    IF (_eMessageLevel = E_MessageType.eMessageVerbose)
    THEN
      _stMsg.eType            := E_MessageType.eMessageVerbose;
      _stMsg.eSubdevice       := e_Subdevice.fbHalt;
      _stMsg.iErrorNumber     := _nErrorId;
      _stMsg.sText            := TO_STRING(_eState);
      f_MessageSet(_stMsg, _nXpu);
    END_IF
END_CASE
//-----------------------------------------------------------------------------
//-----------------------------------------------------------------------------
CASE _eState
OF
  E_PROGRESS.PROGRESS_PREPARE:
    _fbHalt(Axis              := _Mover, 
            Execute           := TRUE, 
            Deceleration      := stMoveData.rAcc, 
            Jerk              := stMoveData.rJerk, 
            BufferMode        := Tc2_MC2.MC_BufferMode.MC_Aborting);

    IF _fbHalt.Error
    THEN
      _bError                 := TRUE;
      _nErrorId               := _fbHalt.ErrorID;
      _eState                 := E_PROGRESS.PROGRESS_ERROR;

      _stMsg.eType            := E_MessageType.eMessageError;
      _stMsg.eSubdevice       := e_Subdevice.fbHalt;
      _stMsg.iErrorNumber     := _nErrorId;
      _stMsg.sText            := TO_STRING(_eState);
      f_MessageSet(_stMsg, _nXpu);

    ELSIF NOT _Mover.Status.Moving
    THEN
      _eState                 := E_PROGRESS.PROGRESS_DONE;

      IF (_eMessageLevel > E_MessageType.eMessageError)
      THEN
        _stMsg.eType          := E_MessageType.eMessageInfo;
        _stMsg.eSubdevice     := e_Subdevice.fbHalt;
        _stMsg.iErrorNumber   := _nErrorId;
        _stMsg.sText          := TO_STRING(_eState);
        f_MessageSet(_stMsg, _nXpu);
      END_IF
    END_IF
END_CASE
//-----------------------------------------------------------------------------
//-----------------------------------------------------------------------------
CASE _eState
OF
  E_PROGRESS.PROGRESS_ERROR,
  E_PROGRESS.PROGRESS_DONE:
    _stInfo.nErrorId          := _nErrorId;
    _fbHalt(
            Axis              := _Mover, 
            Execute           := FALSE);
END_CASE
//-----------------------------------------------------------------------------
//-----------------------------------------------------------------------------

Halt                          := _eState;
END_METHOD

METHOD HaltCa : E_PROGRESS
VAR_INPUT
  Execute             : BOOL;
  stMoveData          : ST_MOVE_DATA;
END_VAR
VAR_INST
  _nErrorId           : UDINT;
  _eState             : E_PROGRESS;
END_VAR
IF NOT Execute 
THEN 
	_eState := E_PROGRESS.PROGRESS_INIT; 
END_IF 
IF NOT Check() 
THEN 
	HaltCa := E_PROGRESS.PROGRESS_ERROR; 
	RETURN; 
END_IF


CASE _eState
OF
  E_PROGRESS.PROGRESS_INIT:
    IF Execute
    THEN
      _nErrorId               := 0;
      _eState                 := E_PROGRESS.PROGRESS_BUSY;
    END_IF
END_CASE
//-----------------------------------------------------------------------------
//-----------------------------------------------------------------------------
CASE _eState
OF
  E_PROGRESS.PROGRESS_BUSY:
    _eState                   := E_PROGRESS.PROGRESS_PREPARE;
    _fbHaltCa(
            Axis              := _Mover, 
            Execute           := FALSE, 
            Deceleration      := stMoveData.rAcc, 
            Jerk              := stMoveData.rJerk, 
            Gap               := stMoveData.rGap);

    IF (_eMessageLevel = E_MessageType.eMessageVerbose)
    THEN
      _stMsg.eType            := E_MessageType.eMessageVerbose;
      _stMsg.eSubdevice       := e_Subdevice.fbHaltCa;
      _stMsg.iErrorNumber     := _nErrorId;
      _stMsg.sText            := TO_STRING(_eState);
      f_MessageSet(_stMsg, _nXpu);
    END_IF
END_CASE
//-----------------------------------------------------------------------------
//-----------------------------------------------------------------------------
CASE _eState
OF
  E_PROGRESS.PROGRESS_PREPARE:
    _fbHaltCa(
            Axis              := _Mover, 
            Execute           := TRUE, 
            Deceleration      := stMoveData.rAcc, 
            Jerk              := stMoveData.rJerk, 
            Gap               := stMoveData.rGap);

    IF _fbHaltCa.Error
    THEN
      _bError                 := TRUE;
      _nErrorId               := _fbHalt.ErrorID;
      _eState                 := E_PROGRESS.PROGRESS_ERROR;

      _stMsg.eType            := E_MessageType.eMessageError;
      _stMsg.eSubdevice       := e_Subdevice.fbHaltCa;
      _stMsg.iErrorNumber     := _nErrorId;
      _stMsg.sText            := TO_STRING(_eState);
      f_MessageSet(_stMsg, _nXpu);

    ELSIF NOT _Mover.Status.Moving
    THEN
      _eState                 := E_PROGRESS.PROGRESS_DONE;

      IF (_eMessageLevel > E_MessageType.eMessageError)
      THEN
        _stMsg.eType          := E_MessageType.eMessageInfo;
        _stMsg.eSubdevice     := e_Subdevice.fbHaltCa;
        _stMsg.iErrorNumber   := _nErrorId;
        _stMsg.sText          := TO_STRING(_eState);
        f_MessageSet(_stMsg, _nXpu);
      END_IF
    END_IF
END_CASE
//-----------------------------------------------------------------------------
//-----------------------------------------------------------------------------
CASE _eState
OF
  E_PROGRESS.PROGRESS_ERROR,
  E_PROGRESS.PROGRESS_DONE:
    _stInfo.nErrorId          := _nErrorId;
    _fbHaltCa(
            Axis              := _Mover, 
            Execute           := FALSE);
END_CASE
//-----------------------------------------------------------------------------
//-----------------------------------------------------------------------------

HaltCa                          := _eState;
END_METHOD

PROPERTY LastGap : REFERENCE to lreal
SET
_rLastGap REF= LastGap;
END_SET
END_PROPERTY

PROPERTY LastPosition : REFERENCE to LREAL
SET
_rLastPosition REF= LastPosition;
END_SET
END_PROPERTY

PROPERTY Master : REFERENCE to AXIS_REF
SET
_Master REF= Master;
END_SET
END_PROPERTY

PROPERTY MessageLevel : e_messagetype
SET
_eMessageLevel := MessageLevel;
END_SET
END_PROPERTY

PROPERTY ModuloTurn : dint
GET
ModuloTurn := _Mover.NcToPlc.ModuloSetTurns;
END_GET
END_PROPERTY

PROPERTY Mover : REFERENCE to AXIS_REF
SET
_Mover REF= Mover;
END_SET
END_PROPERTY

PROPERTY MoverId : uint
SET
_nMoverId := MoverId;
END_SET
END_PROPERTY

PROPERTY MoverInfo : REFERENCE to ST_MOVER_INFO
SET


	_stInfo ref= MoverInfo;
END_SET
END_PROPERTY

METHOD MoveToPos : E_PROGRESS
VAR_INPUT
  Execute             : BOOL;
  stMoveData          : ST_MOVE_DATA;
END_VAR
VAR_INST
  _nErrorId           : UDINT;
  _rDelta,
  _rPos               : LREAL;
  _eState             : E_PROGRESS;
END_VAR
IF NOT Execute THEN _eState  := E_PROGRESS.PROGRESS_INIT; END_IF 
IF NOT Check() THEN MoveToPos   := E_PROGRESS.PROGRESS_ERROR; RETURN; END_IF


CASE _eState
OF
  E_PROGRESS.PROGRESS_INIT:
    IF Execute
    THEN
      _nErrorId               := 0;
      _rDelta                 := SEL((stMoveData.rDelta < 0.01), stMoveData.rDelta, 0.05);
      _eState                 := E_PROGRESS.PROGRESS_BUSY;
    END_IF
END_CASE
//-----------------------------------------------------------------------------
//-----------------------------------------------------------------------------
CASE _eState
OF
  E_PROGRESS.PROGRESS_BUSY:
    _eState                   := E_PROGRESS.PROGRESS_PREPARE;
    _fbPower.Override         := stMoveData.rOverride;

    _rPos                     := ABS(_Mover.NcToPlc.ModuloActTurns)* _RailLength + stMoveData.rPos;


    _rLastPosition            := _rPos;
    //_rLastGap                 := stMoveData.rGap;

    _fbMoveAbs(
            Axis              := _Mover, 
            Execute           := FALSE, 
            Position          := _rPos, 
            Velocity          := stMoveData.rVelo, 
            Acceleration      := stMoveData.rAcc, 
            Deceleration      := stMoveData.rAcc, 
            Jerk              := stMoveData.rJerk, 
            BufferMode        := Tc2_MC2.MC_BufferMode.MC_Aborting);

      IF (_eMessageLevel = E_MessageType.eMessageVerbose)
      THEN
        _stMsg.eType          := E_MessageType.eMessageVerbose;
        _stMsg.eSubdevice     := e_Subdevice.fbMovePtP;
        _stMsg.iErrorNumber   := _nErrorId;
        _stMsg.sText          := concat(TO_STRING(_eState), ': ');
        _stMsg.sText          := concat(_stMsg.sText, concat('stMoveData.rPos: ', TO_STRING(stMoveData.rPos)));
        f_MessageSet(_stMsg, _nXpu);
      END_IF
END_CASE
//-----------------------------------------------------------------------------
//-----------------------------------------------------------------------------
CASE _eState
OF
  E_PROGRESS.PROGRESS_PREPARE:
    _fbMoveAbs(
            Axis              := _Mover, 
            Execute           := TRUE, 
            Position          := _rPos, 
            Velocity          := stMoveData.rVelo, 
            Acceleration      := stMoveData.rAcc, 
            Deceleration      := stMoveData.rAcc, 
            Jerk              := stMoveData.rJerk, 
            BufferMode        := Tc2_MC2.MC_BufferMode.MC_Aborting);

    IF _fbMoveAbs.Error
    THEN
      _bError                 := TRUE;
      _nErrorId               := _fbMoveAbs.ErrorId;
      _eState                 := E_PROGRESS.PROGRESS_ERROR;

      _stMsg.eType            := E_MessageType.eMessageError;
      _stMsg.eSubdevice       := e_Subdevice.fbMovePtP;
      _stMsg.iErrorNumber     := _nErrorId;
      _stMsg.sText            := TO_STRING(_eState);
      f_MessageSet(_stMsg, _nXpu);

    ELSIF _fbMoveAbs.Active OR 
          _fbMoveAbs.Done
		THEN
      _eState                 := E_PROGRESS.PROGRESS_WORKING;

      IF (_eMessageLevel = E_MessageType.eMessageVerbose)
      THEN
        _stMsg.eType          := E_MessageType.eMessageVerbose;
        _stMsg.eSubdevice     := e_Subdevice.fbMovePtP;
        _stMsg.iErrorNumber   := _nErrorId;
        _stMsg.sText          := concat(TO_STRING(_eState), ': ');
        _stMsg.sText          := concat(_stMsg.sText, '.ModuloActPos: ');
        _stMsg.sText          := concat(_stMsg.sText, TO_STRING(_Mover.NcToPlc.ModuloActPos));
        f_MessageSet(_stMsg, _nXpu);
      END_IF
    END_IF
END_CASE
//-----------------------------------------------------------------------------
//-----------------------------------------------------------------------------
CASE _eState
OF
  E_PROGRESS.PROGRESS_WORKING:
    _fbMoveAbs(
          Axis                := _Mover);

    IF _fbMoveAbs.Error
    THEN
      _bError                 := TRUE;
      _nErrorId               := _fbMoveAbs.ErrorId;
      _stInfo.nErrorId        := _nErrorId;
      _eState                 := E_PROGRESS.PROGRESS_ERROR;

      _stMsg.eType            := E_MessageType.eMessageError;
      _stMsg.eSubdevice       := e_Subdevice.fbMovePtP;
      _stMsg.iErrorNumber     := _nErrorId;
      _stMsg.sText            := TO_STRING(_eState);
      f_MessageSet(_stMsg, _nXpu);

      _fbMoveAbs( 
            Axis              := _Mover, 
            Execute           := FALSE);


    ELSIF (_Mover.NcToPlc.ActPos > _fbMoveAbs.Position - _rDelta) AND
          (_Mover.NcToPlc.ActPos < _fbMoveAbs.Position + _rDelta)
    THEN
      IF NOT _Mover.Status.Moving
      THEN
        _eState               := E_PROGRESS.PROGRESS_DONE;

        IF (_eMessageLevel > E_MessageType.eMessageError)
        THEN
          _stMsg.eType        := E_MessageType.eMessageInfo;
          _stMsg.eSubdevice   := e_Subdevice.fbMovePtP;
          _stMsg.iErrorNumber := _nErrorId;
          _stMsg.sText        := concat(TO_STRING(_eState), ': ');
          _stMsg.sText        := concat(_stMsg.sText, concat('ModActPos: ', TO_STRING(_Mover.NcToPlc.ModuloActPos)));
          f_MessageSet(_stMsg, _nXpu);
        END_IF
      _fbMoveAbs( 
            Axis              := _Mover, 
            Execute           := FALSE);
      END_IF
    END_IF
END_CASE
//-----------------------------------------------------------------------------
//-----------------------------------------------------------------------------

MoveToPos                   := _eState;
END_METHOD

METHOD MoveToPosCa : E_PROGRESS
VAR_INPUT
  Execute             : BOOL;
  stMoveData          : ST_MOVE_DATA;
END_VAR
VAR_INST
  _nErrorId           : UDINT;
  _rDelta,
  _rPos               : LREAL;
  _eState             : E_PROGRESS;
END_VAR
IF NOT Execute THEN _eState  := E_PROGRESS.PROGRESS_INIT; END_IF 
IF NOT Check() THEN MoveToPosCa   := E_PROGRESS.PROGRESS_ERROR; RETURN; END_IF


CASE _eState
OF
  E_PROGRESS.PROGRESS_INIT:
    IF Execute
    THEN
      _nErrorId               := 0;
      _rDelta                 := SEL((stMoveData.rDelta < 0.01), stMoveData.rDelta, 0.05);
      _eState                 := E_PROGRESS.PROGRESS_BUSY;
    END_IF
END_CASE
//-----------------------------------------------------------------------------
//-----------------------------------------------------------------------------
CASE _eState
OF
  E_PROGRESS.PROGRESS_BUSY:
    _eState                   := E_PROGRESS.PROGRESS_PREPARE;
    _fbPower.Override         := stMoveData.rOverride;

    _rPos                     := ABS(_Mover.NcToPlc.ModuloActTurns)* _RailLength + stMoveData.rPos;


    _rLastPosition            := _rPos;
    _rLastGap                 := stMoveData.rGap;

    _fbMoveAbsCa( 
            Axis              := _Mover, 
            Execute           := FALSE, 
            ContinuousUpdate  := TRUE, 
            Position          := _rPos,
            Velocity          := stMoveData.rVelo, 
            Acceleration      := stMoveData.rAcc, 
            Deceleration      := stMoveData.rAcc, 
            Jerk              := stMoveData.rJerk, 
            Gap               := stMoveData.rGap, 
            BufferMode        := Tc3_Mc3Definitions.MC_BUFFER_MODE.mcAborting);

    IF (_eMessageLevel = E_MessageType.eMessageVerbose)
    THEN
      _stMsg.eType            := E_MessageType.eMessageVerbose;
      _stMsg.eSubdevice       := e_Subdevice.fbMoveToPosCa;
      _stMsg.iErrorNumber     := _nErrorId;
      _stMsg.sText            := concat(TO_STRING(_eState), ': ');
      _stMsg.sText            := concat(_stMsg.sText, concat('stMoveData.rPos: ', TO_STRING(stMoveData.rPos)));
      f_MessageSet(_stMsg, _nXpu);
    END_IF
END_CASE
//-----------------------------------------------------------------------------
//-----------------------------------------------------------------------------
CASE _eState
OF
  E_PROGRESS.PROGRESS_PREPARE:
    _fbMoveAbsCa( 
            Axis              := _Mover, 
            Execute           := TRUE, 
            ContinuousUpdate  := TRUE, 
            Position          := _rPos,
            Velocity          := stMoveData.rVelo, 
            Acceleration      := stMoveData.rAcc, 
            Deceleration      := stMoveData.rAcc, 
            Jerk              := stMoveData.rJerk, 
            Gap               := stMoveData.rGap, 
            BufferMode        := Tc3_Mc3Definitions.MC_BUFFER_MODE.mcAborting);

    IF _fbMoveAbsCa.Error
    THEN
      _bError                 := TRUE;
      _nErrorId               := _fbMoveAbsCa.ErrorId;
      _stInfo.nErrorId        := _nErrorId;
      _eState                 := E_PROGRESS.PROGRESS_ERROR;

      _stMsg.eType            := E_MessageType.eMessageError;
      _stMsg.eSubdevice       := e_Subdevice.fbMoveToPosCa;
      _stMsg.iErrorNumber     := _nErrorId;
      _stMsg.sText            := TO_STRING(_eState);
      f_MessageSet(_stMsg, _nXpu);

    ELSIF _fbMoveAbsCa.Active OR 
          _fbMoveAbsCa.Done
		THEN
      _eState                 := E_PROGRESS.PROGRESS_WORKING;

      IF (_eMessageLevel = E_MessageType.eMessageVerbose)
      THEN
        _stMsg.eType          := E_MessageType.eMessageVerbose;
        _stMsg.eSubdevice     := e_Subdevice.fbMoveToPosCa;
        _stMsg.iErrorNumber   := _nErrorId;
        _stMsg.sText          := concat(TO_STRING(_eState), ': ');
        _stMsg.sText          := concat(_stMsg.sText, '.ModuloActPos: ');
        _stMsg.sText          := concat(_stMsg.sText, TO_STRING(_Mover.NcToPlc.ModuloActPos));
        f_MessageSet(_stMsg, _nXpu);
      END_IF
    END_IF
END_CASE
//-----------------------------------------------------------------------------
//-----------------------------------------------------------------------------
CASE _eState
OF
  E_PROGRESS.PROGRESS_WORKING:
    _fbMoveAbsCa(
          Axis                := _Mover);

    IF _fbMoveAbsCa.Error
    THEN
      _bError                 := TRUE;
      _nErrorId               := _fbMoveAbsCa.ErrorId;
      _stInfo.nErrorId        := _nErrorId;
      _fbMoveAbsCa( 
            Axis              := _Mover, 
            Execute           := FALSE);

      _eState                 := E_PROGRESS.PROGRESS_ERROR;

      _stMsg.eType            := E_MessageType.eMessageError;
      _stMsg.eSubdevice       := e_Subdevice.fbMoveToPosCa;
      _stMsg.iErrorNumber     := _nErrorId;
      _stMsg.sText            := concat(TO_STRING(_eState), ': ');
      _stMsg.sText            := concat(_stMsg.sText, concat('ModActPos: ', TO_STRING(_Mover.NcToPlc.ModuloActPos)));

      f_MessageSet(_stMsg, _nXpu);

    ELSIF (_Mover.NcToPlc.ActPos > _fbMoveAbsCa.Position - _rDelta) AND
          (_Mover.NcToPlc.ActPos < _fbMoveAbsCa.Position + _rDelta)
    THEN
      IF NOT _Mover.Status.Moving
      THEN
        _eState               := E_PROGRESS.PROGRESS_DONE;

        IF (_eMessageLevel > E_MessageType.eMessageError)
        THEN
          _stMsg.eType        := E_MessageType.eMessageInfo;
          _stMsg.eSubdevice   := e_Subdevice.fbMoveToPosCa;
          _stMsg.iErrorNumber := _nErrorId;
          _stMsg.sText        := concat(TO_STRING(_eState), ': ');
          _stMsg.sText        := concat(_stMsg.sText, concat('ModActPos: ', TO_STRING(_Mover.NcToPlc.ModuloActPos)));
          f_MessageSet(_stMsg, _nXpu);
        END_IF
      _fbMoveAbsCa( 
            Axis              := _Mover, 
            Execute           := FALSE);
      END_IF
    END_IF
END_CASE
//-----------------------------------------------------------------------------
//-----------------------------------------------------------------------------

MoveToPosCa                   := _eState;
END_METHOD

PROPERTY RailLength : LREAL
GET
RailLength := _RailLength;
END_GET
SET
_RailLength := RailLength;
END_SET
END_PROPERTY

METHOD Reset : E_PROGRESS
VAR_INPUT
  Execute             : BOOL;
END_VAR
VAR_INST
  _nErrorId           : UDINT;
  _eState             : E_PROGRESS;
END_VAR
IF NOT Execute THEN _eState  := E_PROGRESS.PROGRESS_INIT; END_IF 
IF NOT Check() THEN Reset    := E_PROGRESS.PROGRESS_ERROR; RETURN; END_IF


CASE _eState
OF
  E_PROGRESS.PROGRESS_INIT:
    IF Execute
    THEN
      _stInfo.nErrorId        :=
      _nErrorId               := 0;
      _eState                 := E_PROGRESS.PROGRESS_BUSY;
    END_IF
END_CASE
//-----------------------------------------------------------------------------
//-----------------------------------------------------------------------------
CASE _eState
OF
  E_PROGRESS.PROGRESS_BUSY:
    _eState                   := E_PROGRESS.PROGRESS_PREPARE;
    _fbReset(
            Axis              := _Mover, 
            Execute           := FALSE);

    IF (_eMessageLevel = E_MessageType.eMessageVerbose)
    THEN
      _stMsg.eType            := E_MessageType.eMessageVerbose;
      _stMsg.eSubdevice       := e_Subdevice.fbReset;
      _stMsg.iErrorNumber     := _nErrorId;
      _stMsg.sText            := TO_STRING(_eState);
      f_MessageSet(_stMsg, _nXpu);
    END_IF
END_CASE
//-----------------------------------------------------------------------------
//-----------------------------------------------------------------------------
CASE _eState
OF
  E_PROGRESS.PROGRESS_PREPARE:
    _fbReset(
            Axis              := _Mover, 
            Execute           := TRUE);

    IF _fbReset.Error
    THEN
      _nErrorId               := _fbReset.ErrorID;
      _eState                 := E_PROGRESS.PROGRESS_ERROR;

      _stMsg.eType            := E_MessageType.eMessageError;
      _stMsg.eSubdevice       := e_Subdevice.fbReset;
      _stMsg.iErrorNumber     := _nErrorId;
      _stMsg.sText            := TO_STRING(_eState);
      f_MessageSet(_stMsg, _nXpu);

    ELSIF NOT _Mover.Status.Moving
    THEN
      _eState                 := E_PROGRESS.PROGRESS_DONE;

      IF (_eMessageLevel > E_MessageType.eMessageError)
      THEN
        _stMsg.eType          := E_MessageType.eMessageInfo;
        _stMsg.eSubdevice     := e_Subdevice.fbReset;
        _stMsg.iErrorNumber   := _nErrorId;
        _stMsg.sText          := TO_STRING(_eState);
        f_MessageSet(_stMsg, _nXpu);
      END_IF
    END_IF
END_CASE
//-----------------------------------------------------------------------------
//-----------------------------------------------------------------------------
CASE _eState
OF
  E_PROGRESS.PROGRESS_ERROR,
  E_PROGRESS.PROGRESS_DONE:
    _stInfo.nErrorId          := _nErrorId;
    _fbReset(
            Axis              := _Mover, 
            Execute           := FALSE);
			
	_bError := FALSE;		
END_CASE
//-----------------------------------------------------------------------------
//-----------------------------------------------------------------------------

Reset                         := _eState;
END_METHOD

METHOD SendToAbsPosCa : E_PROGRESS
VAR_INPUT
  Execute             : BOOL;
  stMoveData          : ST_MOVE_DATA;
END_VAR
VAR_INST
  _nErrorId           : UDINT;
  _rPos               : LREAL;
  _rStart             : LREAL;
  _eState             : E_PROGRESS;
END_VAR
IF NOT Execute THEN _eState  := E_PROGRESS.PROGRESS_INIT; END_IF 
IF NOT Check() THEN SendToAbsPosCa   := E_PROGRESS.PROGRESS_ERROR; RETURN; END_IF


CASE _eState
OF
  E_PROGRESS.PROGRESS_INIT:
    IF Execute
    THEN
      _nErrorId               := 0;
      _rStart                 := _Mover.NcToPlc.ActPos;

      _eState                 := E_PROGRESS.PROGRESS_BUSY;
    END_IF
END_CASE
//-----------------------------------------------------------------------------
//-----------------------------------------------------------------------------
CASE _eState
OF
  E_PROGRESS.PROGRESS_BUSY:
    _eState                   := E_PROGRESS.PROGRESS_PREPARE;
    _fbPower.Override         := stMoveData.rOverride;

    _rPos                     := stMoveData.rPos;
	
    _rLastPosition            := _rPos;
    _rLastGap                 := stMoveData.rGap;

    _fbMoveAbsCa( 
            Axis              := _Mover, 
            Execute           := FALSE, 
            ContinuousUpdate  := TRUE, 
            Position          := _rPos,
            Velocity          := stMoveData.rVelo, 
            Acceleration      := stMoveData.rAcc, 
            Deceleration      := stMoveData.rAcc, 
            Jerk              := stMoveData.rJerk, 
            Gap               := stMoveData.rGap, 
            BufferMode        := Tc3_Mc3Definitions.MC_BUFFER_MODE.mcAborting);

    IF (_eMessageLevel = E_MessageType.eMessageVerbose)
    THEN
      _stMsg.eType            := E_MessageType.eMessageVerbose;
      _stMsg.eSubdevice       := e_Subdevice.fbSendToAbsPosCa;
      _stMsg.iErrorNumber     := _nErrorId;
      _stMsg.sText            := concat(TO_STRING(_eState), ': ');
      _stMsg.sText            := concat(_stMsg.sText, 'stMoveData.rPos: ');
      _stMsg.sText            := concat(_stMsg.sText, TO_STRING(stMoveData.rPos));
      f_MessageSet(_stMsg, _nXpu);

      _stMsg.eType            := E_MessageType.eMessageVerbose;
      _stMsg.eSubdevice       := e_Subdevice.fbSendToAbsPosCa;
      _stMsg.iErrorNumber     := _nErrorId;
      _stMsg.sText            := concat(TO_STRING(_eState), ': ');
      _stMsg.sText            := concat(_stMsg.sText, '.rDistance: ');
      _stMsg.sText            := concat(_stMsg.sText, TO_STRING(stMoveData.rDistance));
      f_MessageSet(_stMsg, _nXpu);
    END_IF
END_CASE
//-----------------------------------------------------------------------------
//-----------------------------------------------------------------------------
CASE _eState
OF
  E_PROGRESS.PROGRESS_PREPARE:
    _fbMoveAbsCa( 
            Axis              := _Mover, 
            Execute           := TRUE, 
            ContinuousUpdate  := TRUE, 
            Position          := _rPos,
            Velocity          := stMoveData.rVelo, 
            Acceleration      := stMoveData.rAcc, 
            Deceleration      := stMoveData.rAcc, 
            Jerk              := stMoveData.rJerk, 
            Gap               := stMoveData.rGap, 
            BufferMode        := Tc3_Mc3Definitions.MC_BUFFER_MODE.mcAborting);

    IF _fbMoveAbsCa.Error
    THEN
      _bError                 := TRUE;
      _nErrorId               := _fbMoveAbsCa.ErrorId;
      _stInfo.nErrorId        := _nErrorId;
      _eState                 := E_PROGRESS.PROGRESS_ERROR;

      _stMsg.eType            := E_MessageType.eMessageError;
      _stMsg.eSubdevice       := e_Subdevice.fbSendToAbsPosCa;
      _stMsg.iErrorNumber     := _nErrorId;
      _stMsg.sText            := TO_STRING(_eState);
      f_MessageSet(_stMsg, _nXpu);

    ELSIF _fbMoveAbsCa.Active OR
          _fbMoveAbsCa.Done
    THEN
      _eState                 := E_PROGRESS.PROGRESS_WORKING;

      IF (_eMessageLevel = E_MessageType.eMessageVerbose)
      THEN
        _stMsg.eType          := E_MessageType.eMessageVerbose;
        _stMsg.eSubdevice     := e_Subdevice.fbSendToAbsPosCa;
        _stMsg.iErrorNumber   := _nErrorId;
        _stMsg.sText          := concat(TO_STRING(_eState), ': ');
        _stMsg.sText          := concat(_stMsg.sText, '.ActPos: ');
        _stMsg.sText          := concat(_stMsg.sText, TO_STRING(_Mover.NcToPlc.ActPos));
        //f_MessageSet(_stMsg, _nXpu);
      END_IF
    END_IF
END_CASE
//-----------------------------------------------------------------------------
//-----------------------------------------------------------------------------
CASE _eState
OF
  E_PROGRESS.PROGRESS_WORKING:
    _fbMoveAbsCa(
            Axis              := _Mover);

    IF _fbMoveAbsCa.Error
    THEN
      _bError                 := TRUE;
      _nErrorId               := _fbMoveAbsCa.ErrorId;
      _stInfo.nErrorId        := _nErrorId;
      _fbMoveAbsCa( 
            Axis              := _Mover, 
            Execute           := FALSE);

      _eState                 := E_PROGRESS.PROGRESS_ERROR;

      _stMsg.eType            := E_MessageType.eMessageError;
      _stMsg.eSubdevice       := e_Subdevice.fbSendToAbsPosCa;
      _stMsg.iErrorNumber     := _nErrorId;
      _stMsg.sText            := TO_STRING(_eState);
      f_MessageSet(_stMsg, _nXpu);

    ELSIF (_Mover.NcToPlc.ActPos > _rStart + stMoveData.rDistance)
    THEN
      _eState                 := E_PROGRESS.PROGRESS_DONE;

      IF (_eMessageLevel > E_MessageType.eMessageError)
      THEN
        _stMsg.eType          := E_MessageType.eMessageInfo;
        _stMsg.eSubdevice     := e_Subdevice.fbSendToAbsPosCa;
        _stMsg.iErrorNumber   := _nErrorId;
        _stMsg.sText          := concat(TO_STRING(_eState), ': ');
        _stMsg.sText          := concat(_stMsg.sText, '.ActPos: ');
        _stMsg.sText          := concat(_stMsg.sText, TO_STRING(_Mover.NcToPlc.ActPos));
        _stMsg.sText          := concat(_stMsg.sText, ' ');
        _stMsg.sText          := concat(_stMsg.sText, '.ActVelo: ');
        _stMsg.sText          := concat(_stMsg.sText, TO_STRING(_Mover.NcToPlc.ActVelo));

        f_MessageSet(_stMsg, _nXpu);
      END_IF
      _fbMoveAbsCa( 
            Axis              := _Mover, 
            Execute           := FALSE);
    END_IF
END_CASE
//-----------------------------------------------------------------------------
//-----------------------------------------------------------------------------

SendToAbsPosCa                := _eState;
END_METHOD

METHOD SendToModuloPosCa : E_PROGRESS
VAR_INPUT
  Execute             : BOOL;
  stMoveData          : ST_MOVE_DATA;
END_VAR
VAR_INST
  _nErrorId           : UDINT;
  _rPos               : LREAL;
  _rStart             : LREAL;
  _eState             : E_PROGRESS;
END_VAR
IF NOT Execute THEN _eState  := E_PROGRESS.PROGRESS_INIT; END_IF 
IF NOT Check() THEN SendToModuloPosCa   := E_PROGRESS.PROGRESS_ERROR; RETURN; END_IF


CASE _eState
OF
  E_PROGRESS.PROGRESS_INIT:
    IF Execute
    THEN
      _nErrorId               := 0;
      _rStart                 := _Mover.NcToPlc.ActPos;

      _eState                 := E_PROGRESS.PROGRESS_BUSY;
    END_IF
    _fbMoveAbsCa( 
          Axis              := _Mover, 
          Execute           := FALSE);
END_CASE
//-----------------------------------------------------------------------------
//-----------------------------------------------------------------------------
CASE _eState
OF
  E_PROGRESS.PROGRESS_BUSY:
    _eState                   := E_PROGRESS.PROGRESS_PREPARE;
    _fbPower.Override         := stMoveData.rOverride;

    _rPos                     := ABS(_Mover.NcToPlc.ModuloActTurns)* _RailLength + stMoveData.rPos;
	
    _rLastPosition            := _rPos;
    _rLastGap                 := stMoveData.rGap;

    _fbMoveAbsCa( 
            Axis              := _Mover, 
            Execute           := FALSE, 
            ContinuousUpdate  := TRUE, 
            Position          := _rPos,
            Velocity          := stMoveData.rVelo, 
            Acceleration      := stMoveData.rAcc, 
            Deceleration      := stMoveData.rAcc, 
            Jerk              := stMoveData.rJerk, 
            Gap               := stMoveData.rGap, 
            BufferMode        := Tc3_Mc3Definitions.MC_BUFFER_MODE.mcAborting);

    IF (_eMessageLevel = E_MessageType.eMessageVerbose)
    THEN
      _stMsg.eType            := E_MessageType.eMessageVerbose;
      _stMsg.eSubdevice       := e_Subdevice.fbSendToModuloPosCa;
      _stMsg.iErrorNumber     := _nErrorId;
      _stMsg.sText            := concat(TO_STRING(_eState), ': ');
      _stMsg.sText            := concat(_stMsg.sText, 'stMoveData.rPos: ');
      _stMsg.sText            := concat(_stMsg.sText, TO_STRING(stMoveData.rPos));
      f_MessageSet(_stMsg, _nXpu);

      _stMsg.eType            := E_MessageType.eMessageVerbose;
      _stMsg.eSubdevice       := e_Subdevice.fbSendToModuloPosCa;
      _stMsg.iErrorNumber     := _nErrorId;
      _stMsg.sText            := concat(TO_STRING(_eState), ': ');
      _stMsg.sText            := concat(_stMsg.sText, '.rDistance: ');
      _stMsg.sText            := concat(_stMsg.sText, TO_STRING(stMoveData.rDistance));
      f_MessageSet(_stMsg, _nXpu);

    END_IF
END_CASE
//-----------------------------------------------------------------------------
//-----------------------------------------------------------------------------
CASE _eState
OF
  E_PROGRESS.PROGRESS_PREPARE:
    _fbMoveAbsCa( 
            Axis              := _Mover, 
            Execute           := TRUE, 
            ContinuousUpdate  := TRUE, 
            Position          := _rPos,
            Velocity          := stMoveData.rVelo, 
            Acceleration      := stMoveData.rAcc, 
            Deceleration      := stMoveData.rAcc, 
            Jerk              := stMoveData.rJerk, 
            Gap               := stMoveData.rGap, 
            BufferMode        := Tc3_Mc3Definitions.MC_BUFFER_MODE.mcAborting);

    IF _fbMoveAbsCa.Error
    THEN
      _bError                 := TRUE;
      _nErrorId               := _fbMoveAbsCa.ErrorId;
      _stInfo.nErrorId        := _nErrorId;
      _eState                 := E_PROGRESS.PROGRESS_ERROR;

      _stMsg.eType            := E_MessageType.eMessageError;
      _stMsg.eSubdevice       := e_Subdevice.fbSendToModuloPosCa;
      _stMsg.iErrorNumber     := _nErrorId;
      _stMsg.sText            := TO_STRING(_eState);
      f_MessageSet(_stMsg, _nXpu);

      _fbMoveAbsCa( 
            Axis              := _Mover, 
            Execute           := FALSE);

    ELSIF _fbMoveAbsCa.Active OR
          _fbMoveAbsCa.Done
    THEN
      _eState                 := E_PROGRESS.PROGRESS_WORKING;

      IF (_eMessageLevel = E_MessageType.eMessageVerbose)
      THEN
        _stMsg.eType          := E_MessageType.eMessageVerbose;
        _stMsg.eSubdevice     := e_Subdevice.fbSendToModuloPosCa;
        _stMsg.iErrorNumber   := _nErrorId;
        _stMsg.sText            := concat(TO_STRING(_eState), ': ');
        _stMsg.sText          := concat(_stMsg.sText, '.ModuloActPos: ');
        _stMsg.sText          := concat(_stMsg.sText, TO_STRING(_Mover.NcToPlc.ModuloActPos));
        //f_MessageSet(_stMsg, _nXpu);
      END_IF
(*
    ELSIF (_Mover.NcToPlc.ActPos > _rStart + stMoveData.rDistance)
    THEN
      _eState                 := E_PROGRESS.PROGRESS_DONE;

      IF (_eMessageLevel < E_MessageType.eMessageError)
      THEN
        _stMsg.eType          := E_MessageType.eMessageInfo;
        _stMsg.eSubdevice     := e_Subdevice.fbSendToModuloPosCa;
        _stMsg.iErrorNumber   := _nErrorId;
        _stMsg.sText          := TO_STRING(_eState);
        f_MessageSet(_stMsg, _nXpu);
      END_IF
      _fbMoveAbsCa( 
            Axis              := _Mover, 
            Execute           := FALSE);
*)
    END_IF
END_CASE
//-----------------------------------------------------------------------------
//-----------------------------------------------------------------------------
CASE _eState
OF
  E_PROGRESS.PROGRESS_WORKING:
    _fbMoveAbsCa(
            Axis              := _Mover);

    IF _fbMoveAbsCa.Error
    THEN
      _bError                 := TRUE;
      _nErrorId               := _fbMoveAbsCa.ErrorId;
      _stInfo.nErrorId        := _nErrorId;
      _fbMoveAbsCa( 
            Axis              := _Mover, 
            Execute           := FALSE);

      _eState                 := E_PROGRESS.PROGRESS_ERROR;

      _stMsg.eType            := E_MessageType.eMessageError;
      _stMsg.eSubdevice       := e_Subdevice.fbSendToModuloPosCa;
      _stMsg.iErrorNumber     := _nErrorId;
      _stMsg.sText            := TO_STRING(_eState);
      f_MessageSet(_stMsg, _nXpu);

    ELSIF (_Mover.NcToPlc.ActPos > _rStart + stMoveData.rDistance)
    THEN
      _eState                 := E_PROGRESS.PROGRESS_DONE;

      IF (_eMessageLevel > E_MessageType.eMessageError)
      THEN
        _stMsg.eType          := E_MessageType.eMessageInfo;
        _stMsg.eSubdevice     := e_Subdevice.fbSendToModuloPosCa;
        _stMsg.iErrorNumber   := _nErrorId;
        _stMsg.sText          := concat(TO_STRING(_eState), ': ');
        _stMsg.sText          := concat(_stMsg.sText, '.ModuloActPos: ');
        _stMsg.sText          := concat(_stMsg.sText, TO_STRING(_Mover.NcToPlc.ModuloActPos));
        _stMsg.sText          := concat(_stMsg.sText, ' ');
        _stMsg.sText          := concat(_stMsg.sText, '.ActVelo: ');
        _stMsg.sText          := concat(_stMsg.sText, TO_STRING(_Mover.NcToPlc.ActVelo));
        f_MessageSet(_stMsg, _nXpu);
      END_IF
      _fbMoveAbsCa( 
            Axis              := _Mover, 
            Execute           := FALSE);
    END_IF
END_CASE
//-----------------------------------------------------------------------------
//-----------------------------------------------------------------------------

SendToModuloPosCa                   := _eState;
END_METHOD

METHOD Stop : E_PROGRESS
VAR_INPUT
  Execute             : BOOL;
  stMoveData          : ST_MOVE_DATA;
END_VAR
VAR_INST
  _nErrorId           : UDINT;
  _eState             : E_PROGRESS;
END_VAR
IF NOT Execute 
THEN 
	_eState := E_PROGRESS.PROGRESS_INIT; 
END_IF 
IF NOT Check() 
THEN 
	Stop := E_PROGRESS.PROGRESS_ERROR; 
	RETURN; 
END_IF


CASE _eState
OF
  E_PROGRESS.PROGRESS_INIT:
    IF Execute
    THEN
      _nErrorId               := 0;
      _eState                 := E_PROGRESS.PROGRESS_BUSY;
    END_IF
END_CASE
//-----------------------------------------------------------------------------
//-----------------------------------------------------------------------------
CASE _eState
OF
  E_PROGRESS.PROGRESS_BUSY:
    _eState                   := E_PROGRESS.PROGRESS_PREPARE;
    _fbStop(
            Axis              := _Mover, 
            Execute           := FALSE, 
            Deceleration      := stMoveData.rAcc, 
            Jerk              := stMoveData.rJerk); 

    IF (_eMessageLevel = E_MessageType.eMessageVerbose)
    THEN
      _stMsg.eType            := E_MessageType.eMessageVerbose;
      _stMsg.eSubdevice       := e_Subdevice.fbStop;
      _stMsg.iErrorNumber     := _nErrorId;
      _stMsg.sText            := TO_STRING(_eState);
      f_MessageSet(_stMsg, _nXpu);
    END_IF
END_CASE
//-----------------------------------------------------------------------------
//-----------------------------------------------------------------------------
CASE _eState
OF
  E_PROGRESS.PROGRESS_PREPARE:
    _fbStop(Axis              := _Mover, 
            Execute           := TRUE, 
            Deceleration      := stMoveData.rAcc, 
            Jerk              := stMoveData.rJerk);

    IF _fbStop.Error
    THEN
      _bError                 := TRUE;
      _nErrorId               := _fbStop.ErrorID;
      _eState                 := E_PROGRESS.PROGRESS_ERROR;

      _stMsg.eType            := E_MessageType.eMessageError;
      _stMsg.eSubdevice       := e_Subdevice.fbStop;
      _stMsg.iErrorNumber     := _nErrorId;
      _stMsg.sText            := TO_STRING(_eState);
      f_MessageSet(_stMsg, _nXpu);

    ELSIF _fbStop.Done
    THEN
      _eState                 := E_PROGRESS.PROGRESS_DONE;

      IF (_eMessageLevel > E_MessageType.eMessageError)
      THEN
        _stMsg.eType          := E_MessageType.eMessageInfo;
        _stMsg.eSubdevice     := e_Subdevice.fbStop;
        _stMsg.iErrorNumber   := _nErrorId;
        _stMsg.sText          := TO_STRING(_eState);
        f_MessageSet(_stMsg, _nXpu);
      END_IF
    END_IF
END_CASE
//-----------------------------------------------------------------------------
//-----------------------------------------------------------------------------
CASE _eState
OF
  E_PROGRESS.PROGRESS_ERROR,
  E_PROGRESS.PROGRESS_DONE:
    _stInfo.nErrorId          := _nErrorId;
    _fbStop(
            Axis              := _Mover, 
            Execute           := FALSE);
END_CASE
//-----------------------------------------------------------------------------
//-----------------------------------------------------------------------------

Stop                          := _eState;
END_METHOD

PROPERTY XpuInstance : uint
SET
//
// Who am I?
// Environment may have more than one ProcessingUnit,
// information required for connecting to the correct instance of ProcessingUnit
_nXpu := XpuInstance;
END_SET
END_PROPERTY

END_FUNCTION_BLOCK

// ---- APPLICATION/MAIN_APP.TcPOU
//---------------------------------------------------------------------------------------------------------------
//
//  HAUD 2024.04.26
//
//  - APPLICATION
//    - explicit simple example PRG for setting up application
//      - no additional interfaces or encapsulations
//      - works dirEctly on GVL_XTS namespace Ctrl/State structs
//      - no error handling, reset application from start
//
//  - Application controls:
//    - XtsTransport
//      - GVL_XTS.TransportCtrl
//      - GVL_XTS.TransportState
//
//    - Xts Stations
//      - GVL_XTS.StationCtrl[]
//      - GVL_XTS.StationState[]
//      - see MAIN.StationParameterInit for XtsStation parameters.
//        - Intention: for developing a transport layer, 
//                      the station parameters are part of the XTS, 
//                      the application primarily handles handshakes with XtsStations
//
//  - Application
//    - 5 single XtsStations
//      - automated handshakes 
//      - process with TON
//      - static targets
//
//---------------------------------------------------------------------------------------------------------------
// This SOFTWARE is provided as an Exemple by THE PROVIDER "as is" and "with all faults." THE PROVIDER makes no 
// representations or warranties of any kind concerning the safety, suitability, lack of viruses, inaccuracies, 
// typographical errors, or other harmful components of this SOFTWARE. There are inherent dangers in the use of 
// any software, and you are solely responsible for determining whether this SOFTWARE is compatible with your 
// equipment and other software installed on your equipment. You are also solely responsible for the protection 
// of your equipment and backup of your data, and THE PROVIDER will not be liable for any damages you may suffer 
// in connection with using, modifying, or distributing this SOFTWARE.
//---------------------------------------------------------------------------------------------------------------
PROGRAM MAIN_APP
VAR
  eInit         : E_PROGRESS;
  bStart        : BOOL;   // XtsTransport is initialized, CAGroup is built, All movers are enabled, XtsStations are cleared, XtsTransport base position for all movers is commanded, XtsStations are handshaked with timer
  bReset        : BOOL;   // All Xts Stations are cleared, requires new start

  nXpu          : UINT;
  nStateError,
  nState        : ARRAY[1..MAX_XPU] OF UINT;   // state var for application

  tonProcess          : ARRAY[1..MAX_XPU] OF ARRAY[1..MAX_STATION] OF Tc2_Standard.TON;
  tProcess            : ARRAY[1..MAX_XPU] OF ARRAY[1..MAX_STATION] OF TIME;

  // work vars
  nStation      : ARRAY[1..MAX_XPU] OF UINT;
  nTarget       : ARRAY[1..MAX_XPU] OF ARRAY[1..MAX_STATION] OF UINT;  // contains target the station is sending the mover to, after process handshake was done

  JobResult     : ARRAY[1..MAX_XPU] OF E_PROGRESS;
END_VAR

//-----------------------------------------------------------------------------
// wait for initialization to be complete before work may start
//-----------------------------------------------------------------------------
IF NOT (Main.eInit = E_PROGRESS.PROGRESS_DONE)
THEN
  eInit                               := E_PROGRESS.PROGRESS_INIT;
  bReset                              := FALSE;
  bStart                              := FALSE;
  memset(ADR(nState), 0, SIZEOF(nState));
  RETURN;
END_IF
//-----------------------------------------------------------------------------
// fetch reset anytime
//-----------------------------------------------------------------------------
IF bReset
THEN
  bReset                              := FALSE;
  bStart                              := FALSE;
  FOR nXpu := 1 TO MAX_XPU
  DO
    nState[nXpu]                      := 9000;  // states for clearing XtsTransport
  END_FOR
END_IF

FOR nXpu := 1 TO MAX_XPU
DO
CASE nState[nXpu] 
OF
  0:                                  // first PLC cycle
    eInit                             := E_PROGRESS.PROGRESS_BUSY;
    nState[nXpu]                      := 1;

    FOR nStation[nXpu] := 1 TO MAX_STATION
    DO
      tProcess[nXpu][nStation[nXpu]]              := T#650MS;
      nTarget [nXpu][nStation[nXpu]]              := SEL(nStation[nXpu]<MAX_STATION, 1, nStation[nXpu]+1);
    END_FOR

  1:
    // do other init stuff here
    eInit                             := E_PROGRESS.PROGRESS_DONE;
    nState[nXpu]                      := 10;

  10:                                 // starts from here
    IF bStart
    THEN
      nStateError[nXpu]               := 0;
      nState[nXpu]                    := 100; // let's go
    END_IF
    
  100:                                // clear interface
    GVL_XTS.XtsTransportCtrl[nXpu].Cmd      := E_XTS_TRANSPORT_CTRL.CMD_NULL;
    nState[nXpu]                            := 110;

  110:                                // check initialization of XtsTransport, wait for either MoverDetection being valid or OperationMode.Simulation
    IF (GVL_XTS.XtsTransportState[nXpu].XpuInfo.IdDetectionValid) OR
       (GVL_XTS.XtsTransportState[nXpu].XpuInfo.OperationMode = OperationMode.Simulation)
    THEN
      // now XtsTransport is initialized, cyclic plausibility checks on Xpu are active
      nState[nXpu]                          := 120;
    END_IF

  120:                                // clear group for defined start situation
    GVL_XTS.XtsTransportCtrl[nXpu].Cmd      := E_XTS_TRANSPORT_CTRL.CMD_GROUP_CLEAR;

    IF (GVL_XTS.XtsTransportState[nXpu].State = E_XTS_TRANSPORT_STATE.TRANSPORT_GROUP_CLEAR + E_PROGRESS.PROGRESS_ERROR)
    THEN
      JobResult[nXpu]                       := GVL_XTS.CaGroupItf[nXpu].McResetAll(FALSE);
      nStateError[nXpu]                     := nState[nXpu];
      nState[nXpu]                          := 9011;

    ELSIF (GVL_XTS.XtsTransportState[nXpu].State = E_XTS_TRANSPORT_STATE.TRANSPORT_GROUP_CLEAR + E_PROGRESS.PROGRESS_DONE)
    THEN
      // CA Group is now in defined error free state
      nState[nXpu]                          := 130;
    END_IF

  130:                                // build Collision Avoidance group with all movers
    GVL_XTS.XtsTransportCtrl[nXpu].Cmd      := E_XTS_TRANSPORT_CTRL.CMD_GROUP_BUILD;

    IF (GVL_XTS.XtsTransportState[nXpu].State = E_XTS_TRANSPORT_STATE.TRANSPORT_GROUP_BUILD + E_PROGRESS.PROGRESS_ERROR)
    THEN
      JobResult[nXpu]                       := GVL_XTS.CaGroupItf[nXpu].McResetAll(FALSE);
      nStateError[nXpu]                     := nState[nXpu];
      nState[nXpu]                          := 9011;

    ELSIF (GVL_XTS.XtsTransportState[nXpu].State = E_XTS_TRANSPORT_STATE.TRANSPORT_GROUP_BUILD + E_PROGRESS.PROGRESS_DONE)
    THEN
      // CA Group contains all movers now
      // GVL_XTS.XtsTransportState.GroupInfo.AxisCount = MAX_MOVER
      nState[nXpu]                          := 140;
    END_IF

  140:                                // enable CA Group
    GVL_XTS.XtsTransportCtrl[nXpu].Cmd      := E_XTS_TRANSPORT_CTRL.CMD_GROUP_ENABLE;

    IF (GVL_XTS.XtsTransportState[nXpu].State = E_XTS_TRANSPORT_STATE.TRANSPORT_GROUP_ENABLE + E_PROGRESS.PROGRESS_ERROR)
    THEN
      JobResult[nXpu]                       := GVL_XTS.CaGroupItf[nXpu].McResetAll(FALSE);
      nStateError[nXpu]                     := nState[nXpu];
      nState[nXpu]                          := 9011;

    ELSIF (GVL_XTS.XtsTransportState[nXpu].State = E_XTS_TRANSPORT_STATE.TRANSPORT_GROUP_ENABLE + E_PROGRESS.PROGRESS_DONE)
    THEN
      // GVL_XTS.XtsTransportState.GroupInfo.CaGroupState = mcGroupStateNotReady
      nState[nXpu]                          := 150;
    END_IF

  150:                                // enable all movers
    GVL_XTS.XtsTransportCtrl[nXpu].Cmd      := E_XTS_TRANSPORT_CTRL.CMD_MOVER_ENABLE;

    IF (GVL_XTS.XtsTransportState[nXpu].State = E_XTS_TRANSPORT_STATE.TRANSPORT_MOVER_ENABLE + E_PROGRESS.PROGRESS_ERROR)
    THEN
      JobResult[nXpu]                       := GVL_XTS.CaGroupItf[nXpu].McResetAll(FALSE);
      nStateError[nXpu]                     := nState[nXpu];
      nState[nXpu]                          := 9011;

    ELSIF (GVL_XTS.XtsTransportState[nXpu].State = E_XTS_TRANSPORT_STATE.TRANSPORT_MOVER_ENABLE + E_PROGRESS.PROGRESS_DONE)
    THEN
      // GVL_XTS.XtsTransportState.GroupInfo.CaGroupState = mcGroupStateStandby
      nState[nXpu]                          := 160;
    END_IF

  160:                                // command all movers to startup position
    GVL_XTS.XtsTransportCtrl[nXpu].Cmd      := E_XTS_TRANSPORT_CTRL.CMD_TRANSPORT_START;

    IF (GVL_XTS.XtsTransportState[nXpu].State = E_XTS_TRANSPORT_STATE.TRANSPORT_START + E_PROGRESS.PROGRESS_DONE)
    THEN
      // all XtsStations are cleared
      // all movers are now waiting at GVL_XTS.XtsTransport.StartStationIndex
      // all movers are entered into GVL_XTS.StationList[GVL_XTS.XtsTransport.StartStationIndex]._stList 
      nState[nXpu]                          := 170;
    END_IF

  170:
    nState[nXpu]                            := 1000;

  1000:                               // automatic handshakes with XtsStations
    FOR nStation[nXpu] := 1 TO MAX_STATION
    DO
      CASE GVL_XTS.StationState[nXpu][nStation[nXpu]].eState
      OF
        E_STATION_STATE.STATION_DISABLE:          // switch on XtsStation
          GVL_XTS.StationCtrl[nXpu][nStation[nXpu]].eCmd      := E_STATION_CTRL.STATION_ENABLE;

        E_STATION_STATE.STATION_MOVER_ENTER:      // let mover enter
          // mover was detected in list and station is asking for mover entry
          GVL_XTS.StationCtrl[nXpu][nStation[nXpu]].eCmd      := E_STATION_CTRL.STATION_MOVER_ENTER;  // allow entry
          //GVL_XTS.StationCtrl[nStation].eCmd      := E_STATION_CTRL.STATION_MOVER_SEND;  // no process handshake, direct state change to MOVER_OUT 

        E_STATION_STATE.STATION_PROCESS_START:    // first process handshake, clear timer
          // mover has arrived and is in standstill, ready for process 
          tonProcess[nXpu][nStation[nXpu]](
                              IN                  :=FALSE, 
                              PT                  :=tProcess[nXpu][nStation[nXpu]]);
          GVL_XTS.StationCtrl[nXpu][nStation[nXpu]].eCmd      := E_STATION_CTRL.STATION_PROCESS_START;

        E_STATION_STATE.STATION_PROCESS_DONE:     // second process handshake, timer runs now
          tonProcess[nXpu][nStation[nXpu]](
                              IN                  :=TRUE, 
                              PT                  :=tProcess[nXpu][nStation[nXpu]]);
          IF tonProcess[nXpu][nStation[nXpu]].Q
          THEN
            GVL_XTS.StationCtrl[nXpu][nStation[nXpu]].eCmd    := E_STATION_CTRL.STATION_PROCESS_DONE;
          END_IF

        E_STATION_STATE.STATION_MOVER_OUT:        // station wants to send out mover
          // when sending out mover, the data on Ctrl struct is absolute important
          // before allowing the outfeed of the mover, the data on Ctrl struct must be entered correctly
          // Ctrl.nTargetStation allows for flexible mover transport, this is fully depending on you to make sense aside this example

          GVL_XTS.StationCtrl[nXpu][nStation[nXpu]].nTargetStation  := TO_USINT(nTarget[nXpu][nStation[nXpu]]); // static in this example
          GVL_XTS.StationCtrl[nXpu][nStation[nXpu]].nMask     := 2#1; // bitmask for mover ticket to next XtsStation; if you use more than one StopPos[] in XtsStation

          GVL_XTS.StationCtrl[nXpu][nStation[nXpu]].eCmd      := E_STATION_CTRL.STATION_MOVER_OUT;  // allow outfeed of mover

        E_STATION_STATE.STATION_MOVER_GONE:       // mover has travelled ReleaseDistance, XtsStation is now empty and ready for the next mover in queue
          GVL_XTS.StationCtrl[nXpu][nStation[nXpu]].nTargetStation  := 0;                           // clear target after mover left the station
          GVL_XTS.StationCtrl[nXpu][nStation[nXpu]].eCmd      := E_STATION_CTRL.STATION_MOVER_GONE; // last handshake for empty station
      END_CASE
    END_FOR


  9000:
    GVL_XTS.XtsTransportCtrl[nXpu].Cmd      := E_XTS_TRANSPORT_CTRL.CMD_NULL;
    nState[nXpu]                            := 9010;

  9010:                               // halt all movers and clear group
    GVL_XTS.XtsTransportCtrl[nXpu].Cmd      := E_XTS_TRANSPORT_CTRL.CMD_GROUP_CLEAR;

    IF (GVL_XTS.XtsTransportState[nXpu].State = E_XTS_TRANSPORT_STATE.TRANSPORT_GROUP_CLEAR + E_PROGRESS.PROGRESS_ERROR)
    THEN
      JobResult[nXpu]                       := GVL_XTS.CaGroupItf[nXpu].McResetAll(FALSE);
      nState[nXpu]                          := 9011;

    ELSIF (GVL_XTS.XtsTransportState[nXpu].State = E_XTS_TRANSPORT_STATE.TRANSPORT_GROUP_CLEAR + E_PROGRESS.PROGRESS_DONE)
    THEN
      // CA group cleared and mover in standstill
      nState[nXpu]                          := 9100;
    END_IF

  9011:
    JobResult[nXpu]                         := GVL_XTS.CaGroupItf[nXpu].McResetAll(TRUE);

    IF (JobResult[nXpu] = E_PROGRESS.PROGRESS_DONE)
    THEN
      nState[nXpu]                          := 9012;
      JobResult[nXpu]                       := GVL_XTS.CaGroupItf[nXpu].McResetAll(FALSE);
      JobResult[nXpu]                       := GVL_XTS.CaGroupItf[nXpu].Reset(FALSE);
    END_IF

  9012:
    JobResult[nXpu]                         := GVL_XTS.CaGroupItf[nXpu].Reset(TRUE);

    IF (JobResult[nXpu] = E_PROGRESS.PROGRESS_DONE)
    THEN
      nState[nXpu]                          := 9000;
      JobResult[nXpu]                       := GVL_XTS.CaGroupItf[nXpu].Reset(FALSE);
    END_IF


  9100:                               // switch off movers
    GVL_XTS.XtsTransportCtrl[nXpu].Cmd      := E_XTS_TRANSPORT_CTRL.CMD_MOVER_DISABLE;

    IF (GVL_XTS.XtsTransportState[nXpu].State >= E_XTS_TRANSPORT_STATE.TRANSPORT_MOVER_DISABLE + E_PROGRESS.PROGRESS_ERROR)
    THEN
      nState[nXpu]                          := 9200;
    END_IF

  9200:                               // clear All XtsStations
    nState[nXpu]                            := 9300;
    FOR nStation[nXpu] := 1 TO MAX_STATION
    DO
       GVL_XTS.StationCtrl[nXpu][nStation[nXpu]].eCmd      := E_STATION_CTRL.STATION_INIT;
    END_FOR

  9300:                               // disable All XtsStations
    nState[nXpu]                            := 10;   // go back to start
    FOR nStation[nXpu] := 1 TO MAX_STATION
    DO
       GVL_XTS.StationCtrl[nXpu][nStation[nXpu]].eCmd      := E_STATION_CTRL.STATION_DISABLE;
    END_FOR
END_CASE
END_FOR

END_PROGRAM

// ---- MAIN.TcPOU
//---------------------------------------------------------------------------------------------------------------
//
//  HAUD 2024.03.18
//
//  - XTS_TRANSPORT_LAYER
//  - transport layer members:
//    - CaGroup
//      - access to Group functions
//
//    - Mover
//      - access to MC and CA motion functions
//
//    - Xpu (ProcessingUnit)
//      - access to TcCOM Objects in Environment
//
//    - Transport Control Unit
//      - coordinates members to get XTS in defined states
//
//    - Xts Stations
//      - handshakes with extern control for mover transport
//
//  - global datafields for mrmbers in GVL_XTS namespace
//  - global interface datafields for use in members
//  - structures are assigned by reference for every member
//
//---------------------------------------------------------------------------------------------------------------
// HAUD 2024 05 29
//
//    XTS_TRANSPORT_LAYER project
//    
//    MIT License
//    
//    Copyright (c) 2024 HAUD
//    
//    Permission is hereby granted, free of charge, to any person obtaining a copy
//    of this software and associated documentation files (the "Software"), to deal
//    in the Software without restriction, including without limitation the rights
//    to use, copy, modify, merge, publish, distribute, sublicense, and/or sell
//    copies of the Software, and to permit persons to whom the Software is
//    furnished to do so, subject to the following conditions:
//    
//    The above copyright notice and this permission notice shall be included in all
//    copies or substantial portions of the Software.
//    
//    THE SOFTWARE IS PROVIDED "AS IS", WITHOUT WARRANTY OF ANY KIND, EXPRESS OR
//    IMPLIED, INCLUDING BUT NOT LIMITED TO THE WARRANTIES OF MERCHANTABILITY,
//    FITNESS FOR A PARTICULAR PURPOSE AND NONINFRINGEMENT. IN NO EVENT SHALL THE
//    AUTHORS OR COPYRIGHT HOLDERS BE LIABLE FOR ANY CLAIM, DAMAGES OR OTHER
//    LIABILITY, WHETHER IN AN ACTION OF CONTRACT, TORT OR OTHERWISE, ARISING FROM,
//    OUT OF OR IN CONNECTION WITH THE SOFTWARE OR THE USE OR OTHER DEALINGS IN THE
//    SOFTWARE.
//---------------------------------------------------------------------------------------------------------------
PROGRAM MAIN
VAR
	bInit 				: BOOL;
  eInit         : E_PROGRESS;
  wInit         : DWORD;

  nXpu,
  nXpuSelected,
  nStation,
	nMover,
  nMoverSelected,
  nStationSelected,
  nStationParameter   : UINT;

  sStationText        : STRING(30);

  eTransportState     : E_XTS_TRANSPORT_STATE;
  eTransportResult    : E_PROGRESS;

  eXpuState           : E_XPU_STATE;
  eXpuResult          : E_PROGRESS;
  eXpuCheck           : E_XPU_CHECK;

  eMoverState         : E_MOVER_STATE;
  eMoverResult        : E_PROGRESS;

  sCaGroupState,
  sTransportState,
  sTransportCheck,
  sTransportResult,
  sXpuState,
  sXpuResult,
  sXpuCheck,
  sXpuOpMode,
  sXpuMoverdetectionMode,
  sXpuMoverAssignement,
  sMoverState,
  sMoverResult,
  sStationState,
  sStationStateMask,
  sStationCtrlMask        : STRING;

  bStationEnable,
  bStationEnter,
  bStationStart,
  bStationDone,
  bStationOut,
  bStationGone            : BOOL;

  tStationSelectedQueue   : ARRAY[1..MAX_LIST_NODES] OF ST_STATION_MOVER_DATA;

  tonWriteLog             : ARRAY[1..MAX_XPU] OF Tc2_Standard.TON;
  tWriteLog               : TIME := T#5S;
END_VAR

//############################################################################
// Local time; used for timestamps
//############################################################################
GVL_MSG.fbLocalTime(
                    sLocalTime          => GVL_MSG.sLocalTime, 
                    dtLocalTime         => GVL_MSG.dtLocalTime);
//############################################################################

//############################################################################
// 	example for init sequence
//############################################################################	
IF NOT bInit
THEN
  CASE eInit
  OF
    E_PROGRESS.PROGRESS_INVALID,
    E_PROGRESS.PROGRESS_DONE:         // clear command interface
      wInit                                   := 0;
      eInit                                   := E_PROGRESS.PROGRESS_BUSY;
      FOR nXpu := 1 TO MAX_XPU
      DO
        GVL_XTS.XpuCtrl[nXpu].Cmd             := E_XPU_CTRL.XTS_CMD_NULL;
        GVL_MSG.MessageLevelXpu               := GVL_MSG.MessageLevel;
        GVL_XTS.CaGroup[nXpu].MessageLevel    := GVL_MSG.MessageLevel;

        FOR nStation := 1 TO MAX_STATION
        DO
          GVL_MSG.MessageLevelStations[nXpu][nStation]:= GVL_MSG.MessageLevel;
        END_FOR
        FOR nMover := 1 TO MAX_MOVER
        DO
          GVL_MSG.MessageLevelMovers[nXpu][nMover]    := GVL_MSG.MessageLevel;
        END_FOR
      END_FOR

    E_PROGRESS.PROGRESS_BUSY:         // init Xpu, ProcessingUnit, MotorModules
      GVL_XTS.XpuCtrl[1].Cmd                  := E_XPU_CTRL.XTS_CMD_INIT;

      IF (GVL_XTS.XpuState[1].State      = E_XPU_STATE.XTS_INIT + E_PROGRESS.PROGRESS_DONE)
      THEN
        wInit := Tc2_System.SETBIT32(wInit, TO_SINT(1-1));
        eInit                                 := E_PROGRESS.PROGRESS_PREPARE;
      END_IF


    E_PROGRESS.PROGRESS_PREPARE:      // wait for init to be done
      GVL_XTS.XpuCtrl[2].Cmd                  := E_XPU_CTRL.XTS_CMD_INIT;
      IF (GVL_XTS.XpuState[2].State      = E_XPU_STATE.XTS_INIT + E_PROGRESS.PROGRESS_DONE)
      THEN
        wInit := Tc2_System.SETBIT32(wInit, TO_SINT(2-1));
      END_IF

      IF (wInit = TO_DWORD(EXPT(2,MAX_XPU))-1)
      THEN
        eInit                                 := E_PROGRESS.PROGRESS_STARTUP;
      END_IF

    E_PROGRESS.PROGRESS_STARTUP:      // assign mover interfaces
      eInit                                   := E_PROGRESS.PROGRESS_CHECK;
      FOR nXpu := 1 TO MAX_XPU
      DO
        GVL_XTS.XpuCtrl[nXpu].Cmd             := E_XPU_CTRL.XTS_IDLE;
        FOR nMover := 1 TO MAX_MOVER
        DO
          GVL_XTS.MoverItf[nXpu][nMover]      := GVL_XTS.Mover[nXpu][nMover];
        END_FOR
      END_FOR


    E_PROGRESS.PROGRESS_CHECK:        // assign CaGroup interface
      eInit                                   := E_PROGRESS.PROGRESS_OCCUPIED;
      GVL_XTS.CaGroupItf[nXpu]                := GVL_XTS.CaGroup[nXpu];

    E_PROGRESS.PROGRESS_OCCUPIED:     // StartStation for XtsTransportCtrl.Cmd := E_XTS_TRANSPORT_CTRL.CMD_TRANSPORT_START;
      eInit                                   := E_PROGRESS.PROGRESS_WORKING;
      // where to start?

      // Start Position parameters
      GVL_XTS.StationStart[1].rPosWait           :=     10.0;
      GVL_XTS.StationStart[1].rGap               :=    150.0;
      GVL_XTS.StationStart[1].rVelo              :=   1250.0;
      GVL_XTS.StationStart[1].rAccDec            :=  12000.0;
      GVL_XTS.StationStart[1].rJerk              := 400000.0;
      GVL_XTS.XtsTransport[1].StationStartIndex  := 1;

      // Start Position parameters
      GVL_XTS.StationStart[2].rPosWait           :=     10.0;
      GVL_XTS.StationStart[2].rGap               :=    150.0;
      GVL_XTS.StationStart[2].rVelo              :=   1250.0;
      GVL_XTS.StationStart[2].rAccDec            :=  12000.0;
      GVL_XTS.StationStart[2].rJerk              := 400000.0;
      GVL_XTS.XtsTransport[2].StationStartIndex  := 1;

    E_PROGRESS.PROGRESS_WORKING:
      // hard coded XTS Station parameter are here:
      StationParameterInit();

      // initialization of XtsTransport is done here:
      bInit                                   := TRUE;
      eInit                                   := E_PROGRESS.PROGRESS_DONE;
  END_CASE
END_IF

//############################################################################
// 	XTS Transport Unit
//############################################################################
//  - main control function block for transport layer
//  - requires access to member controls
//    - Xpu
//    - CaGroup
//    - Mover
//    - Station Control
//    - Station LinkedList Interface
//############################################################################
//
// cyclic call
FOR nXpu := 1 TO MAX_XPU
DO
  GVL_XTS.XtsTransport[nXpu].XpuInstance        := nXpu;

  GVL_XTS.XtsTransport[nXpu]();
  
  // main control
  GVL_XTS.XtsTransport[nXpu].Ctrl               REF= GVL_XTS.XtsTransportCtrl[nXpu];   // main control
  GVL_XTS.XtsTransport[nXpu].State              REF= GVL_XTS.XtsTransportState[nXpu];  // main state
                                          
  // member controls                      
  GVL_XTS.XtsTransport[nXpu].XpuCtrl            REF= GVL_XTS.XpuCtrl[nXpu];
  GVL_XTS.XtsTransport[nXpu].XpuState           REF= GVL_XTS.XpuState[nXpu];
  GVL_XTS.XtsTransport[nXpu].XpuInfo            REF= GVL_XTS.XpuInfo[nXpu];
                                          
  GVL_XTS.XtsTransport[nXpu].GroupItf           :=   GVL_XTS.CaGroupItf[nXpu];
  GVL_XTS.XtsTransport[nXpu].GroupInfo          REF= GVL_XTS.CaGroupInfo[nXpu];
                                          
  GVL_XTS.XtsTransport[nXpu].MoverItf           REF= GVL_XTS.MoverItf[nXpu];
  GVL_XTS.XtsTransport[nXpu].MoverInfo          REF= GVL_XTS.MoverInfo[nXpu];
  GVL_XTS.XtsTransport[nXpu].MoverLastPosition  REF= GVL_XTS.LastPosition[nXpu];
  GVL_XTS.XtsTransport[nXpu].MoverLastGap       REF= GVL_XTS.LastGap[nXpu];
                                          
  GVL_XTS.XtsTransport[nXpu].StationStart       REF= GVL_XTS.StationStart[nXpu];      // start position for E_XTS_TRANSPORT_CTRL.CMD_TRANSPORT_START
  GVL_XTS.XtsTransport[nXpu].StationCtrlItf     REF= GVL_XTS.StationCtrlItf[nXpu];    // station interfaces are required for accessing station methods
  GVL_XTS.XtsTransport[nXpu].StationListsItf    REF= GVL_XTS.StationListItf[nXpu];    // list interface is required for access to linked list methods
  GVL_XTS.XtsTransport[nXpu].StationControl     REF= GVL_XTS.StationCtrl[nXpu];
  GVL_XTS.XtsTransport[nXpu].StationState       REF= GVL_XTS.StationState[nXpu];
  //############################################################################
  
  
  
  //############################################################################
  // 	XTS Stations
  //############################################################################	
  FOR nStation := 1 TO MAX_STATION
  DO
    GVL_XTS.Station[nXpu][nStation].XpuInstance := nXpu;
    GVL_XTS.Station[nXpu][nStation].StationId   := nStation;
    GVL_XTS.Station[nXpu][nStation].MessageLevel:= GVL_MSG.MessageLevelStations[nXpu][nStation];
  
    GVL_XTS.StationListItf[nXpu][nStation]      := GVL_XTS.StationList[nXpu][nStation];   // interfaces for list methods
    GVL_XTS.StationCtrlItf[nXpu][nStation]      := GVL_XTS.Station[nXpu][nStation];       // interfaces for station methods
  
    GVL_XTS.Station[nXpu][nStation].Ctrl        REF= GVL_XTS.StationCtrl[nXpu];           // station ctrl from extern
    GVL_XTS.Station[nXpu][nStation].State       REF= GVL_XTS.StationState[nXpu];          // station state to extern
  
    GVL_XTS.Station[nXpu][nStation].ItfStations REF= GVL_XTS.StationListItf[nXpu];        // give every station all list interfaces for writing mover tickets
    GVL_XTS.Station[nXpu][nStation].ItfMover    REF= GVL_XTS.MoverItf[nXpu];              // give every station all mover interfaces for movement in / out of station
    GVL_XTS.Station[nXpu][nStation].Mover       REF= GVL_XTS.AxisRefMover[nXpu];          // AXIS_REF to read infos from
    GVL_XTS.Station[nXpu][nStation].MoverOffset REF= GVL_XTS.PositionOffset[nXpu];        // static offsets for all stations, all movers, all stop positions
  
  
    GVL_XTS.Station[nXpu][nStation].StationParameter  REF= GVL_XTS.StationParameter[nXpu];// give every station all station parameters for sending to WaitPos of target station
  
    // cyclic call
    GVL_XTS.Station[nXpu][nStation].Cycle();                                        // cycle for handshaking with extern
  
    // Queue data for each station
    GVL_XTS.StationQueue[nXpu][nStation]        := GVL_XTS.StationListItf[nXpu][nStation].Data;
  END_FOR
  //############################################################################
  
  
  
  //############################################################################
  // 	XPU environment
  //############################################################################	
  GVL_XTS.Xpu[nXpu].XpuInstance               :=   nXpu;
  GVL_XTS.Xpu[nXpu].MessageLevel              :=   GVL_MSG.MessageLevelXpu;
  
  GVL_XTS.Xpu[nXpu].Ctrl                      REF= GVL_XTS.XpuCtrl[nXpu];
  GVL_XTS.Xpu[nXpu].State                     REF= GVL_XTS.XpuState[nXpu];
  GVL_XTS.Xpu[nXpu].XpuModuleInfoData         REF= GVL_XTS.XpuModules[nXpu];
  
  GVL_XTS.Xpu[nXpu].CaGroupOID                :=   GVL_XTS.CaGroup[nXpu].GroupInfo.CaGroupOID;
  
  // cyclic call
  GVL_XTS.Xpu[nXpu]();
  GVL_XTS.XpuInfo[nXpu]                       :=   GVL_XTS.Xpu[nXpu].XpuInfo;
  //############################################################################
  
  
  //############################################################################	
  // 	CA-Group Class
  //############################################################################
  GVL_XTS.CaGroup[nXpu].XpuInstance           := nXpu; // for every XPU there must be a CA group in this example	
  // assignment
  GVL_XTS.CaGroup[nXpu].AxisRef               REF= GVL_XTS.AxisRefMover[nXpu];
  // Interface to Mover methods
  GVL_XTS.CaGroup[nXpu].MoverItf              REF= GVL_XTS.MoverItf[nXpu]; 
  
  GVL_XTS.CaGroup[nXpu].GroupRef              REF= GVL_XTS.CaGroupRef[nXpu];
  
  // cyclic call
  GVL_XTS.CaGroup[nXpu].InfoCycle(TRUE); // read group status
  
  // InfoData from group
  GVL_XTS.CaGroupInfo[nXpu]                   :=   GVL_XTS.CaGroup[nXpu].GroupInfo;
  
  // Interface of CaGroup
  GVL_XTS.CaGroupItf[nXpu]                    :=   GVL_XTS.CaGroup[nXpu];
  //############################################################################
  
  
  //############################################################################
  // Mover Class	
  //############################################################################	
  FOR nMover := 1 TO MAX_MOVER
  DO
    GVL_XTS.Mover[nXpu][nMover].XpuInstance   :=   nXpu;
    GVL_XTS.Mover[nXpu][nMover].MoverId       :=   nMover;
    GVL_XTS.Mover[nXpu][nMover].RailLength    :=   GVL_XTS.Xpu[nXpu].RailLength;  // mover needs RailLength, in order to calc absolute position from modulo input
    GVL_XTS.Mover[nXpu][nMover].MessageLevel  :=   GVL_MSG.MessageLevelMovers[nXpu][nMover];
  
    GVL_XTS.Mover[nXpu][nMover].Ctrl          REF= GVL_XTS.MoverCtrl[nXpu];       // mover control from extern
    GVL_XTS.Mover[nXpu][nMover].State         REF= GVL_XTS.MoverState[nXpu];      // mover state to extern
  
    GVL_XTS.Mover[nXpu][nMover].MoveData      REF= GVL_XTS.MoveData[nXpu];        // dyn constraints for extern to write
    GVL_XTS.Mover[nXpu][nMover].GearData      REF= GVL_XTS.GearData[nXpu];        // GearIn/GearInPosCa data fro extern to write
  
    // assignment	
    GVL_XTS.Mover[nXpu][nMover].Mover         REF= GVL_XTS.AxisRefMover[nXpu][nMover];  // axis reference to Mover function block
    GVL_XTS.Mover[nXpu][nMover].LastGap       REF= GVL_XTS.LastGap[nXpu][nMover];       // reference to last used gap value datafield
    GVL_XTS.Mover[nXpu][nMover].LastPosition  REF= GVL_XTS.LastPosition[nXpu][nMover];  // reference to last position datafield
  
    GVL_XTS.Mover[nXpu][nMover].MoverInfo		  REF= GVL_XTS.MoverInfo[nXpu][nMover];     // refernence to mover info data (ActPos, SetPos, ...)
  
    GVL_XTS.MoverItf[nXpu][nMover]            :=   GVL_XTS.Mover[nXpu][nMover];
  
    // cyclic call
    GVL_XTS.Mover[nXpu][nMover].Cycle();  // call AXIS_REF()
    GVL_XTS.Mover[nXpu][nMover]();        // call Ctrl/State
  END_FOR
  //############################################################################
  // /logging
  //############################################################################
  tonWriteLog[nXpu](IN:= TRUE, PT := tWriteLog);
  
  IF (tonWriteLog[nXpu].Q)
  THEN
    GVL_MSG.MessageData[nXpu].bWriteFile      := TRUE;
    tonWriteLog[nXpu](IN:= FALSE);
  END_IF
  
  //-----------------------------------------------------------------------------------------------------------------
  // write message list to file
  //-----------------------------------------------------------------------------------------------------------------
  GVL_MSG.MessageData[nXpu](
              pList			        := ADR(GVL_MSG.Messages[nXpu]),
              pLocalTime        := ADR(GVL_MSG.dtLocalTime),
              nXpu              := nXpu,
              bBusy=> );
  
  // clear write trigger
  IF GVL_MSG.MessageData[nXpu].bWriteFile AND
     GVL_MSG.MessageData[nXpu].bDone
  THEN
    GVL_MSG.MessageData[nXpu].bWriteFile      := FALSE;
  END_IF
  //############################################################################
  // logging/
  //############################################################################
END_FOR

//############################################################################
//############################################################################
// Visualization data	
//############################################################################	
nXpuSelected                          := SEL((nXpuSelected<1), nXpuSelected, 1);
nXpuSelected                          := SEL((nXpuSelected>MAX_XPU), nXpuSelected, MAX_XPU);
// get enumerations from XPU for visu:
eTransportState                       := f_GetState   (GVL_XTS.XtsTransportState[nXpuSelected].State);
eTransportResult                      := f_GetProgress(GVL_XTS.XtsTransportState[nXpuSelected].State);

eXpuState                             := f_GetState   (GVL_XTS.XpuState[nXpuSelected].State);
eXpuResult                            := f_GetProgress(GVL_XTS.XpuState[nXpuSelected].State);

eXpuCheck                             := GVL_XTS.XpuState[nXpuSelected].Check;

// display xpu state and result in visu
// get strings and info
sCaGroupState                         := TO_STRING(GVL_XTS.CaGroupInfo[nXpuSelected].CaGroupState);

sTransportState                       := TO_STRING(eTransportState);
sTransportCheck                       := TO_STRING(GVL_XTS.XtsTransportState[nXpuSelected].Check);
sTransportResult                      := TO_STRING(eTransportResult);

sXpuState                             := TO_STRING(eXpuState);
sXpuResult                            := TO_STRING(eXpuResult);
sXpuCheck                             := TO_STRING(eXpuCheck);

sXpuOpMode                            := GVL_XTS.Xpu[nXpuSelected].OpModeToString();
sXpuMoverdetectionMode                := GVL_XTS.Xpu[nXpuSelected].IdDetectionModeToString();
sXpuMoverAssignement                  := GVL_XTS.Xpu[nXpuSelected].MoverPositionAssignementToString();

nMoverSelected                        := SEL((nMoverSelected<1), nMoverSelected, 1);
nMoverSelected                        := SEL((nMoverSelected>MAX_MOVER), nMoverSelected, MAX_MOVER);

nStationSelected                      := SEL((nStationSelected<1), nStationSelected, 1);
nStationSelected                      := SEL((nStationSelected>MAX_STATION), nStationSelected, MAX_STATION);

bStationEnable                        := SEL((GVL_XTS.StationCtrl[nXpuSelected][nStationSelected].eCmd = E_STATION_CTRL.STATION_ENABLE),        FALSE, TRUE);
bStationEnter                         := SEL((GVL_XTS.StationCtrl[nXpuSelected][nStationSelected].eCmd = E_STATION_CTRL.STATION_MOVER_ENTER),   FALSE, TRUE);
bStationStart                         := SEL((GVL_XTS.StationCtrl[nXpuSelected][nStationSelected].eCmd = E_STATION_CTRL.STATION_PROCESS_START), FALSE, TRUE);
bStationDone                          := SEL((GVL_XTS.StationCtrl[nXpuSelected][nStationSelected].eCmd = E_STATION_CTRL.STATION_PROCESS_DONE),  FALSE, TRUE);
bStationOut                           := SEL((GVL_XTS.StationCtrl[nXpuSelected][nStationSelected].eCmd = E_STATION_CTRL.STATION_MOVER_OUT),     FALSE, TRUE);
bStationGone                          := SEL((GVL_XTS.StationCtrl[nXpuSelected][nStationSelected].eCmd = E_STATION_CTRL.STATION_MOVER_GONE),    FALSE, TRUE);

eMoverState                           := f_GetState   (GVL_XTS.MoverState[nXpuSelected][nMoverSelected].State);
eMoverResult                          := f_GetProgress(GVL_XTS.MoverState[nXpuSelected][nMoverSelected].State);

sMoverState                           := TO_STRING(eMoverState);
sMoverResult                          := TO_STRING(eMoverResult);

sStationState                         := TO_STRING(GVL_XTS.StationState[nXpuSelected][nStationSelected].eState);
sStationStateMask                     := Tc2_Utilities.BYTE_TO_BINSTR(GVL_XTS.StationState[nXpuSelected][nStationSelected].nMask, 8);
sStationCtrlMask                      := Tc2_Utilities.BYTE_TO_BINSTR(GVL_XTS.StationCtrl[nXpuSelected][nStationSelected].nMask, 8);

tStationSelectedQueue                 := GVL_XTS.StationQueue[nXpuSelected][nStationSelected];

ACTION StationParameterInit:
//-----------------------------------------------------------------------------
//
//  HAUD 2025.08.18
//
//  - hard coded station parameters as example
//  - TODO: xml DataServer implementation for station parameter read/write
//
//  - reminder: (this you HAVE to check manually when setting up the transport)
//-----------------------------------------------------------------------------
//    - DO NOT place the modulo turn within the range of a station
//
//    - in case the extern process requires multiple xts stations, 
//      - the range must be closed and in strict order
//-----------------------------------------------------------------------------
//-----------------------------------------------------------------------------

FOR nXpu := 1 TO MAX_XPU
DO
  //-----------------------------------------------------------------------------------------------------------------------------------------
  nStationParameter := 1;
  GVL_XTS.StationParameter[nXpu][nStationParameter].rPosWait              :=    140.0; // absolute modulo position
  
  GVL_XTS.StationParameter[nXpu][nStationParameter].nConfiguredStopCount  :=      1;   // how many stops the mover has to make in this station
  GVL_XTS.StationParameter[nXpu][nStationParameter].rPosStop[1]           :=    235.0; // relative to rPosWait
  
  GVL_XTS.StationParameter[nXpu][nStationParameter].rReleaseDistance      :=     75.0; // relative to Mover.ActPos
  
  GVL_XTS.StationParameter[nXpu][nStationParameter].rGap                  :=    105.0;
  GVL_XTS.StationParameter[nXpu][nStationParameter].rVelo                 :=   1250.0;
  GVL_XTS.StationParameter[nXpu][nStationParameter].rAccDec               :=  17500.0;
  GVL_XTS.StationParameter[nXpu][nStationParameter].rJerk                 := 600000.0;
  
  //-----------------------------------------------------------------------------------------------------------------------------------------
  nStationParameter := 2;
  GVL_XTS.StationParameter[nXpu][nStationParameter].rPosWait              :=   1890.0; // absolute modulo position
  
  GVL_XTS.StationParameter[nXpu][nStationParameter].nConfiguredStopCount  :=      1;   // how many stops the mover has to make in this station
  GVL_XTS.StationParameter[nXpu][nStationParameter].rPosStop[1]           :=    235.0; // relative to rPosWait
  
  GVL_XTS.StationParameter[nXpu][nStationParameter].rReleaseDistance      :=    350.0; // relative to Mover.ActPos
  
  GVL_XTS.StationParameter[nXpu][nStationParameter].rGap                  :=    105.0;
  GVL_XTS.StationParameter[nXpu][nStationParameter].rVelo                 :=   1250.0;
  GVL_XTS.StationParameter[nXpu][nStationParameter].rAccDec               :=  17500.0;
  GVL_XTS.StationParameter[nXpu][nStationParameter].rJerk                 := 600000.0;
  
  //-----------------------------------------------------------------------------------------------------------------------------------------
  nStationParameter := 3;
  GVL_XTS.StationParameter[nXpu][nStationParameter].rPosWait              :=   2640.0; // absolute modulo position
  
  GVL_XTS.StationParameter[nXpu][nStationParameter].nConfiguredStopCount  :=      1;   // how many stops the mover has to make in this station
  GVL_XTS.StationParameter[nXpu][nStationParameter].rPosStop[1]           :=    235.0; // relative to rPosWait
  
  GVL_XTS.StationParameter[nXpu][nStationParameter].rReleaseDistance      :=    150.0; // relative to Mover.ActPos
  
  GVL_XTS.StationParameter[nXpu][nStationParameter].rGap                  :=    105.0;
  GVL_XTS.StationParameter[nXpu][nStationParameter].rVelo                 :=   1500.0;
  GVL_XTS.StationParameter[nXpu][nStationParameter].rAccDec               :=  17500.0;
  GVL_XTS.StationParameter[nXpu][nStationParameter].rJerk                 := 600000.0;
  
  //-----------------------------------------------------------------------------------------------------------------------------------------
  nStationParameter := 4;
  GVL_XTS.StationParameter[nXpu][nStationParameter].rPosWait              :=   3640.0; // absolute modulo position
  
  GVL_XTS.StationParameter[nXpu][nStationParameter].nConfiguredStopCount  :=      1;   // how many stops the mover has to make in this station
  GVL_XTS.StationParameter[nXpu][nStationParameter].rPosStop[1]           :=    235.0; // relative to rPosWait
  
  GVL_XTS.StationParameter[nXpu][nStationParameter].rReleaseDistance      :=    100.0; // relative to Mover.ActPos
  
  GVL_XTS.StationParameter[nXpu][nStationParameter].rGap                  :=    105.0;
  GVL_XTS.StationParameter[nXpu][nStationParameter].rVelo                 :=   1500.0;
  GVL_XTS.StationParameter[nXpu][nStationParameter].rAccDec               :=  17500.0;
  GVL_XTS.StationParameter[nXpu][nStationParameter].rJerk                 := 600000.0;
  
  //-----------------------------------------------------------------------------------------------------------------------------------------
  nStationParameter := 5;
  GVL_XTS.StationParameter[nXpu][nStationParameter].rPosWait              :=   4890.0; // absolute modulo position
  
  GVL_XTS.StationParameter[nXpu][nStationParameter].nConfiguredStopCount  :=      1;   // how many stops the mover has to make in this station
  GVL_XTS.StationParameter[nXpu][nStationParameter].rPosStop[1]           :=    235.0; // relative to rPosWait
  
  GVL_XTS.StationParameter[nXpu][nStationParameter].rReleaseDistance      :=     50.0; // relative to Mover.ActPos
  
  GVL_XTS.StationParameter[nXpu][nStationParameter].rGap                  :=    105.0;
  GVL_XTS.StationParameter[nXpu][nStationParameter].rVelo                 :=   1500.0;
  GVL_XTS.StationParameter[nXpu][nStationParameter].rAccDec               :=  17500.0;
  GVL_XTS.StationParameter[nXpu][nStationParameter].rJerk                 := 600000.0;
END_FOR
END_ACTION

END_PROGRAM

// ---- GlobalTextList.TcGTLO
TEXTLIST GlobalTextList
  17 = ' STATION_ENABLE'
  34 = ' STATION_MOVER_ENTER'
  452 = ' STATION_MOVER_GONE'
  75 = ' STATION_MOVER_OUT'
  598 = ' STATION_PROCESS_DONE'
  750 = ' STATION_PROCESS_START'
  294 = '%.2f'
  191 = '%d'
  836 = '%s'
  248 = 'Activate'
  444 = 'Activate Visu list'
  704 = 'All Positions Valid'
  562 = 'AllAxisStanding'
  878 = 'AxisCount Enabled: %d'
  162 = 'AxisCount: %d'
  914 = 'ConstantVelocity'
  929 = 'Control'
  707 = 'CyclicCheck: %s'
  660 = 'DC Link All Modules'
  359 = 'Decelerating'
  843 = 'Detected AxisCount: %d'
  243 = 'eDevice'
  244 = 'eSubdevice'
  242 = 'eType'
  772 = 'Expected AxisCount: %d'
  48 = 'GroupDisabled'
  915 = 'GroupError'
  495 = 'GroupErrorId: %d'
  975 = 'GroupErrorStop'
  940 = 'GroupHoming'
  300 = 'GroupMoving'
  807 = 'GroupNotReady'
  438 = 'GroupStandby'
  226 = 'GroupStatusBusy'
  204 = 'GroupStatusValid'
  973 = 'GroupStopping'
  942 = 'GVL_XTS.CaGroupInfo'
  680 = 'ID Detection Active'
  238 = 'ID Detection Error'
  526 = 'ID Detection Mode: %s'
  29 = 'ID Detection Valid'
  245 = 'iErrorNumber'
  211 = 'Info Act Pos Absolute'
  586 = 'Info Act Pos Modulo'
  21 = 'Info Mover Avoiding Collision'
  282 = 'Info Mover Coupled'
  398 = 'Info Mover Enabled'
  751 = 'Info Mover Error'
  907 = 'Info Mover Standstill'
  480 = 'Info nError ID'
  922 = 'Info Target Pos Absolute'
  16 = 'Info Target Pos Modulo'
  616 = 'InPosition'
  713 = 'Mask: %b'
  972 = 'Mask: %d'
  779 = 'Mask: %s'
  726 = 'McGroupState:      %s'
  160 = 'McGroupState: %d  %s'
  974 = 'MOVER command'
  387 = 'Mover ID: %d'
  297 = 'Mover Position Assignement: %s'
  840 = 'MOVER result:  %s'
  53 = 'MOVER state:   %s'
  756 = 'nMoverSelected: %d'
  669 = 'nStation selected: %d'
  94 = 'Offset %.3f'
  427 = 'Offset: %.3f'
  312 = 'Operation Mode: %s'
  320 = 'Queue: %d'
  91 = 'Set Acceleration'
  399 = 'Set Delta'
  382 = 'Set Distance'
  757 = 'Set Gap'
  934 = 'Set Jerk'
  201 = 'Set Override'
  936 = 'Set Position'
  62 = 'Set Velocity'
  231 = 'State'
  748 = 'Station Control'
  267 = 'Station State'
  627 = 'STATION_ENABLE'
  247 = 'sText'
  54 = 'Target Station %d'
  567 = 'Target Station: %d'
  246 = 'tTime'
  517 = 'WRITE TO FILE'
  541 = 'XPU (selected): %d'
  275 = 'XPU Command'
  227 = 'XpuResult:   %s'
  96 = 'XpuState:    %s'
  43 = 'XTS (selected): %d'
  884 = 'XTS Station'
  572 = 'XTS Transport Check:  %s'
  212 = 'XTS Transport Check: %s'
  500 = 'XTS Transport Command'
  395 = 'XTS Transport Result: %s'
  798 = 'XTS Transport State:  %s'
  417 = 'XTS Transport State: %s'
END_TEXTLIST

// ---- XTS/_Visualization/GROUP_VISU.TcVIS
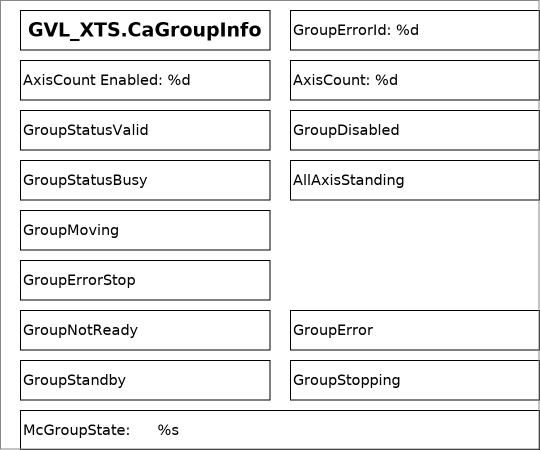
VISUALIZATION GROUP_VISU  // 540x450
    Rectangle (20,110 250x40), "GroupStatusValid", colour toggle: GVL_XTS.XtsTransportState[MAIN.nXpuSelected].GroupInfo.GroupStatusValid
    Rectangle (20,160 250x40), "GroupStatusBusy", colour toggle: GVL_XTS.XtsTransportState[MAIN.nXpuSelected].GroupInfo.GroupStatusBusy
    Rectangle (20,210 250x40), "GroupMoving", colour toggle: GVL_XTS.XtsTransportState[MAIN.nXpuSelected].GroupInfo.GroupMoving
    Rectangle (20,260 250x40), "GroupErrorStop", colour toggle: GVL_XTS.XtsTransportState[MAIN.nXpuSelected].GroupInfo.GroupErrorStop
    Rectangle (20,310 250x40), "GroupNotReady", colour toggle: GVL_XTS.XtsTransportState[MAIN.nXpuSelected].GroupInfo.GroupNotReady
    Rectangle (20,360 250x40), "GroupStandby", colour toggle: GVL_XTS.XtsTransportState[MAIN.nXpuSelected].GroupInfo.GroupStandby
    Rectangle (290,360 250x40), "GroupStopping", colour toggle: GVL_XTS.XtsTransportState[MAIN.nXpuSelected].GroupInfo.GroupStopping
    Rectangle (290,110 250x40), "GroupDisabled", colour toggle: GVL_XTS.XtsTransportState[MAIN.nXpuSelected].GroupInfo.GroupDisabled
    Rectangle (290,160 250x40), "AllAxisStanding", colour toggle: GVL_XTS.XtsTransportState[MAIN.nXpuSelected].GroupInfo.AllAxesStanding
    Rectangle (290,310 250x40), "GroupError", colour toggle: GVL_XTS.XtsTransportState[MAIN.nXpuSelected].GroupInfo.GroupError
    Rectangle (290,10 250x40), "GroupErrorId: %d", text variable: GVL_XTS.XtsTransportState[MAIN.nXpuSelected].GroupInfo.GroupErrorId
    Rectangle (290,60 250x40), "AxisCount: %d", text variable: GVL_XTS.XtsTransportState[MAIN.nXpuSelected].GroupInfo.AxisCount
    Rectangle (20,410 520x40), "McGroupState: %s", text variable: MAIN.sCaGroupState
    Rectangle (20,10 250x40), "GVL_XTS.CaGroupInfo"
    Rectangle (20,60 250x40), "AxisCount Enabled: %d", text variable: GVL_XTS.CaGroupInfo[MAIN.nXpuSelected].AxisCountEnabled
END_VISUALIZATION

// ---- XTS/_Visualization/XTS_TRANSPORT.TcVIS
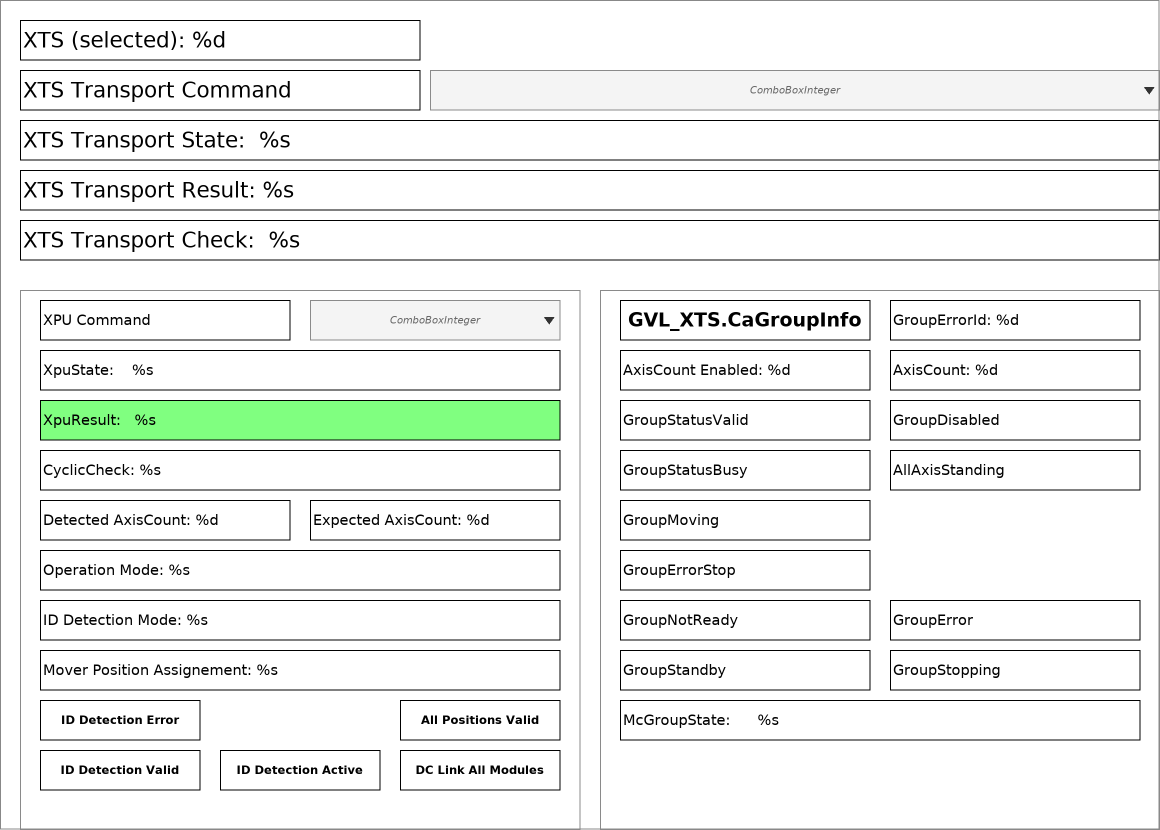
VISUALIZATION XTS_TRANSPORT  // 1160x830
    Rectangle (20,70 400x40), "XTS Transport Command"
    ComboBoxInteger (430,70 730x40), variable: GVL_XTS.XtsTransportCtrl[MAIN.nXpuSelected].Cmd, text list: 'TL_E_CTRL_TRANSPORT'
    Frame (20,290 560x540)
        shows XPU_VISU()
    Frame (600,290 560x540)
        shows GROUP_VISU()
    Rectangle (20,120 1140x40), "XTS Transport State: %s", text variable: MAIN.sTransportState
    Rectangle (20,170 1140x40), "XTS Transport Result: %s", text variable: MAIN.sTransportResult
    Rectangle (20,220 1140x40), "XTS Transport Check: %s", text variable: MAIN.sTransportCheck
    Rectangle (20,20 400x40), "XTS (selected): %d", text variable: MAIN.nXpuSelected
        OnMouseClick: write the text variable via VisuDialogs.Numpad, min 1, max MAX_XPU, title 'Select XPU'
END_VISUALIZATION

// ---- XTS/_Visualization/XPU_VISU.TcVIS
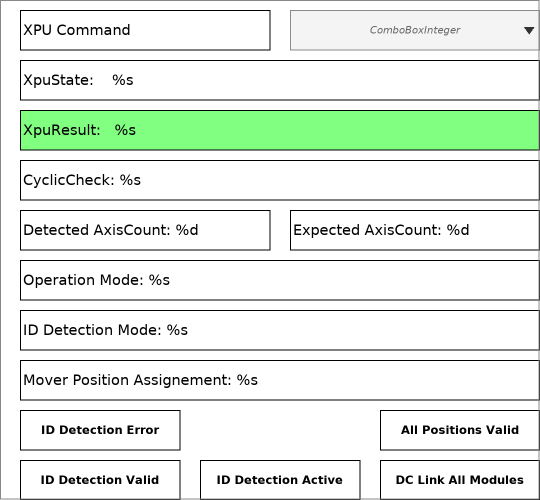
VISUALIZATION XPU_VISU  // 540x500
    Rectangle (20,10 250x40), "XPU Command"
    ComboBoxInteger (290,10 250x40), variable: GVL_XTS.XpuCtrl[MAIN.nXpuSelected].Cmd, text list: 'TL_E_CTRL_XPU'
    Rectangle (20,160 520x40), "CyclicCheck: %s", text variable: MAIN.sXpuCheck
    Rectangle (20,60 520x40), "XpuState: %s", text variable: MAIN.sXpuState
    Rectangle (20,110 520x40), "XpuResult: %s", text variable: MAIN.sXpuResult, colour toggle: (MAIN.eXpuResult = E_PROGRESS.PROGRESS_ERROR)
    Rectangle (380,410 160x40), "All Positions Valid", colour toggle: GVL_XTS.XtsTransportState[MAIN.nXpuSelected].XpuInfo.AllPositionsValid
    Rectangle (20,410 160x40), "ID Detection Error", colour toggle: GVL_XTS.XtsTransportState[MAIN.nXpuSelected].XpuInfo.IdDetectionError
    Rectangle (20,460 160x40), "ID Detection Valid", colour toggle: GVL_XTS.XtsTransportState[MAIN.nXpuSelected].XpuInfo.IdDetectionValid
    Rectangle (200,460 160x40), "ID Detection Active", colour toggle: GVL_XTS.XtsTransportState[MAIN.nXpuSelected].XpuInfo.IdDetectionActive
    Rectangle (20,260 520x40), "Operation Mode: %s", text variable: MAIN.sXpuOpMode
    Rectangle (20,310 520x40), "ID Detection Mode: %s", text variable: MAIN.sXpuMoverdetectionMode
    Rectangle (20,360 520x40), "Mover Position Assignement: %s", text variable: MAIN.sXpuMoverAssignement
    Rectangle (290,210 250x40), "Expected AxisCount: %d", text variable: GVL_XTS.XtsTransportState[MAIN.nXpuSelected].XpuInfo.nExpectedAxisCount
    Rectangle (20,210 250x40), "Detected AxisCount: %d", text variable: GVL_XTS.XtsTransportState[MAIN.nXpuSelected].XpuInfo.nDetectedAxisCount
    Rectangle (380,460 160x40), "DC Link All Modules", colour toggle: GVL_XTS.XtsTransportState[MAIN.nXpuSelected].XpuState.DcLink
END_VISUALIZATION
